	{attribute 'TcIecLibraryType'}
	{attribute 'external_name' := 'F_VN_ImageAverageStdDevExp_GUID_F60066E2_6F02_44CC_C0FB_3753E15EF1D8'}
	(* Computes the (channel-wise) average pixel value and the corresponding standard deviation of an image. (expert function) *)
	FUNCTION F_VN_ImageAverageStdDevExp : HRESULT
	VAR_INPUT
		ipSrcImage	:	ITcVnImage;	(* Source image (1 - 4 channels) *)
	END_VAR
	VAR_IN_OUT
		aAverage	:	TcVnVector4_LREAL;	(* Returns the (channel-wise) average pixel value of ipSrcImage *)
		aStdDev	:	TcVnVector4_LREAL;	(* Returns the (channel-wise) pixel value standard deviation of ipSrcImage *)
	END_VAR
	VAR_INPUT
		ipMask	:	ITcVnImage;	(* Mask of type USINT (1 channel) *)
		hrPrev	:	HRESULT;	(* HRESULT indicating the result of previous operations (If SUCCEEDED(hrPrev) equals false, no operation is executed.) *)
	END_VAR

END_FUNCTION

// Functions/Image Analysis/F_VN_ImageCenterOfMass

	{attribute 'TcIecLibraryType'}
	{attribute 'external_name' := 'F_VN_ImageCenterOfMass_GUID_92F451E2_12EA_4476_D35C_66DCB9E907BA'}
	(* Computes the center of mass of an image. *)
	FUNCTION F_VN_ImageCenterOfMass : HRESULT
	VAR_INPUT
		ipSrcImage	:	ITcVnImage;	(* Source image (1 channel) *)
	END_VAR
	VAR_IN_OUT
		aCenterOfMass	:	TcVnPoint2_LREAL;	(* Returns the center of mass of the image *)
	END_VAR
	VAR_INPUT
		hrPrev	:	HRESULT;	(* HRESULT indicating the result of previous operations (If SUCCEEDED(hrPrev) equals false, no operation is executed.) *)
	END_VAR

END_FUNCTION

// Functions/Image Analysis/F_VN_ImageCenterOfMassExp

	{attribute 'TcIecLibraryType'}
	{attribute 'external_name' := 'F_VN_ImageCenterOfMassExp_GUID_2975F517_49B1_4459_C14B_04840D9F0255'}
	(* Computes the center of mass of an image. *)
	FUNCTION F_VN_ImageCenterOfMassExp : HRESULT
	VAR_INPUT
		ipSrcImage	:	ITcVnImage;	(* Source image (1 channel) *)
	END_VAR
	VAR_IN_OUT
		aCenterOfMass	:	TcVnPoint2_LREAL;	(* Returns the center of mass of the image *)
	END_VAR
	VAR_INPUT
		ipMask	:	ITcVnImage;	(* Optional mask (1 channel of type USINT, same width and height as ipSrcImage) *)
		hrPrev	:	HRESULT;	(* HRESULT indicating the result of previous operations (If SUCCEEDED(hrPrev) equals false, no operation is executed.) *)
	END_VAR

END_FUNCTION

// Functions/Image Analysis/F_VN_ImageMedian

	{attribute 'TcIecLibraryType'}
	{attribute 'external_name' := 'F_VN_ImageMedian_GUID_8462A627_DBC4_4874_EF70_B1418DB7E2BB'}
	(* Computes the (approximated, channel-wise) median pixel value of an image. *)
	FUNCTION F_VN_ImageMedian : HRESULT
	VAR_INPUT
		ipSrcImage	:	ITcVnImage;	(* Source image (1 - 4 channels) *)
	END_VAR
	VAR_IN_OUT
		aMedian	:	TcVnVector4_LREAL;	(* Returns the (approximated, channel-wise) median pixel value of ipSrcImage *)
	END_VAR
	VAR_INPUT
		hrPrev	:	HRESULT;	(* HRESULT indicating the result of previous operations (If SUCCEEDED(hrPrev) equals false, no operation is executed.) *)
	END_VAR

END_FUNCTION

// Functions/Image Analysis/F_VN_ImageMedianExp

	{attribute 'TcIecLibraryType'}
	{attribute 'external_name' := 'F_VN_ImageMedianExp_GUID_04A4F1B3_1CC2_4D44_C68C_989FB7E7D270'}
	(* Computes the (approximated, channel-wise) median pixel value of an image. (expert function) *)
	FUNCTION F_VN_ImageMedianExp : HRESULT
	VAR_INPUT
		ipSrcImage	:	ITcVnImage;	(* Source image (1 - 4 channels) *)
	END_VAR
	VAR_IN_OUT
		aMedian	:	TcVnVector4_LREAL;	(* Returns the (approximated, channel-wise) median pixel value of ipSrcImage *)
	END_VAR
	VAR_INPUT
		ipMask	:	ITcVnImage;	(* Mask of type USINT (1 channel) *)
		hrPrev	:	HRESULT;	(* HRESULT indicating the result of previous operations (If SUCCEEDED(hrPrev) equals false, no operation is executed.) *)
	END_VAR

END_FUNCTION

// Functions/Image Analysis/F_VN_ImageMoments

	{attribute 'TcIecLibraryType'}
	{attribute 'external_name' := 'F_VN_ImageMoments_GUID_967E76E1_3BDD_4152_E4CB_6D63F11261EF'}
	(* Computes the spatial moments, the central moments, and the central normalized moments of an image up to the third order. *)
	FUNCTION F_VN_ImageMoments : HRESULT
	VAR_INPUT
		ipImage	:	ITcVnImage;	(* Source image (1 channel, elements of type USINT or REAL) *)
	END_VAR
	VAR_IN_OUT
		stMoments	:	TcVnMoments;	(* Returns a struct containing the moments *)
	END_VAR
	VAR_INPUT
		bBinaryImage	:	BOOL;	(* If true, all non-zero pixels are treated as ones *)
		hrPrev	:	HRESULT;	(* HRESULT indicating the result of previous operations (If SUCCEEDED(hrPrev) equals false, no operation is executed.) *)
	END_VAR

END_FUNCTION

// Functions/Image Analysis/F_VN_MaxPixelValue

	{attribute 'TcIecLibraryType'}
	{attribute 'external_name' := 'F_VN_MaxPixelValue_GUID_413B82D5_F755_40D2_D677_A4C5ED7EF55F'}
	(* Finds the maximum pixel value in an image (1 - 4 channels supported). *)
	FUNCTION F_VN_MaxPixelValue : HRESULT
	VAR_INPUT
		ipImage	:	ITcVnImage;	(* Source image *)
	END_VAR
	VAR_IN_OUT
		aMaxValue	:	TcVnVector4_LREAL;	(* Returns the maximum pixel value *)
		aPosition	:	TcVnPoint2_DINT;	(* Returns the first found position of aMaxValue *)
	END_VAR
	VAR_INPUT
		hrPrev	:	HRESULT;	(* HRESULT indicating the result of previous operations (If SUCCEEDED(hrPrev) equals false, no operation is executed.) *)
	END_VAR

END_FUNCTION

// Functions/Image Analysis/F_VN_MaxPixelValueExp

	{attribute 'TcIecLibraryType'}
	{attribute 'external_name' := 'F_VN_MaxPixelValueExp_GUID_6DE06A3E_73A8_4932_DDB7_AC3625332A92'}
	(* Finds the maximum pixel value in an image (1 - 4 channels supported). (expert function) *)
	FUNCTION F_VN_MaxPixelValueExp : HRESULT
	VAR_INPUT
		ipImage	:	ITcVnImage;	(* Source image *)
	END_VAR
	VAR_IN_OUT
		aMaxValue	:	TcVnVector4_LREAL;	(* Returns the maximum pixel value *)
		aPosition	:	TcVnPoint2_DINT;	(* Returns the first found position of aMaxValue (not supported for multi-channel images with ELEMENTWISE) *)
	END_VAR
	VAR_INPUT
		ipMask	:	ITcVnImage;	(* Optional mask to specify which pixel positions are considered (USINT, set parameter to 0 if not required) *)
		eVectorCompareMethod	:	ETcVnVectorCompareMethod;	(* Select a vector compare method for multi-channel images *)
		hrPrev	:	HRESULT;	(* HRESULT indicating the result of previous operations (If SUCCEEDED(hrPrev) equals false, no operation is executed.) *)
	END_VAR

END_FUNCTION

// Functions/Image Analysis/F_VN_MinPixelValue

	{attribute 'TcIecLibraryType'}
	{attribute 'external_name' := 'F_VN_MinPixelValue_GUID_2CD718DC_24E2_49FF_F186_BB52705C26CA'}
	(* Finds the minimum pixel value in an image (1 - 4 channels supported). *)
	FUNCTION F_VN_MinPixelValue : HRESULT
	VAR_INPUT
		ipImage	:	ITcVnImage;	(* Source image *)
	END_VAR
	VAR_IN_OUT
		aMinValue	:	TcVnVector4_LREAL;	(* Returns the minimum pixel value *)
		aPosition	:	TcVnPoint2_DINT;	(* Returns the first found position of aMinValue *)
	END_VAR
	VAR_INPUT
		hrPrev	:	HRESULT;	(* HRESULT indicating the result of previous operations (If SUCCEEDED(hrPrev) equals false, no operation is executed.) *)
	END_VAR

END_FUNCTION

// Functions/Image Analysis/F_VN_MinPixelValueExp

	{attribute 'TcIecLibraryType'}
	{attribute 'external_name' := 'F_VN_MinPixelValueExp_GUID_F4A5D3CA_6503_48EC_C514_4486EF0B3DEE'}
	(* Finds the minimum pixel value in an image (1 - 4 channels supported). (expert function) *)
	FUNCTION F_VN_MinPixelValueExp : HRESULT
	VAR_INPUT
		ipImage	:	ITcVnImage;	(* Source image *)
	END_VAR
	VAR_IN_OUT
		aMinValue	:	TcVnVector4_LREAL;	(* Returns the minimum pixel value *)
		aPosition	:	TcVnPoint2_DINT;	(* Returns the first found position of aMinValue (not supported for multi-channel images with ELEMENTWISE) *)
	END_VAR
	VAR_INPUT
		ipMask	:	ITcVnImage;	(* Optional mask to specify which pixel positions are considered (USINT, set parameter to 0 if not required) *)
		eVectorCompareMethod	:	ETcVnVectorCompareMethod;	(* Select a vector compare method for multi-channel images *)
		hrPrev	:	HRESULT;	(* HRESULT indicating the result of previous operations (If SUCCEEDED(hrPrev) equals false, no operation is executed.) *)
	END_VAR

END_FUNCTION

// Functions/Image Analysis/F_VN_RegionOrientation

	{attribute 'TcIecLibraryType'}
	{attribute 'external_name' := 'F_VN_RegionOrientation_GUID_40AE352D_EC33_486F_FD9D_BE6F8D8BC7EF'}
	(* Calculate the orientation of a region based on a binary image that contains a non zero value for every pixel in that region. *)
	FUNCTION F_VN_RegionOrientation : HRESULT
	VAR_INPUT
		ipSrcImage	:	ITcVnImage;	(* Source image (1 channel, binary). *)
	END_VAR
	VAR_IN_OUT
		stOrientation	:	TcVnRotatedRectangle;	(* Resulting rotated rectangle, containig center of mass, lenghts of axes, and rotation angle of the region in clockwise direction. *)
	END_VAR
	VAR_INPUT
		hrPrev	:	HRESULT;	(* HRESULT indicating the result of previous operations (If SUCCEEDED(hrPrev) equals false, no operation is executed.) *)
	END_VAR

END_FUNCTION

// Functions/Image Analysis/F_VN_RegionOrientationExp

	{attribute 'TcIecLibraryType'}
	{attribute 'external_name' := 'F_VN_RegionOrientationExp_GUID_5D1BC303_88B3_462A_E97C_3FA0A9CBE9C1'}
	(* Calculate the orientation of a region based on a binary image that contains a non zero value for every pixel in that region. (expert function) *)
	FUNCTION F_VN_RegionOrientationExp : HRESULT
	VAR_INPUT
		ipSrcImage	:	ITcVnImage;	(* Source image (1 channel, binary) *)
	END_VAR
	VAR_IN_OUT
		stOrientation	:	TcVnRotatedRectangle;	(* Resulting rotated rectangle, containig center of mass, lenghts of axes, and rotation angle of the region in clockwise direction. *)
	END_VAR
	VAR_INPUT
		eMethod	:	ETcVnOrientationMethod;	(* Method for calculating the orientation. *)
		hrPrev	:	HRESULT;	(* HRESULT indicating the result of previous operations (If SUCCEEDED(hrPrev) equals false, no operation is executed.) *)
	END_VAR

END_FUNCTION

// Functions/Image Analysis/F_VN_UprightInnerRectangle

	{attribute 'TcIecLibraryType'}
	{attribute 'external_name' := 'F_VN_UprightInnerRectangle_GUID_EAF07AE8_844F_488F_C920_29FB31213543'}
	(* Computes the maximum area upright inner rectangle inside an area. If the valid area contains very small invalid areas or the performance is too slow, use the expert variant of this function and manually choose a suitable nDownScaleFactor. *)
	FUNCTION F_VN_UprightInnerRectangle : HRESULT
	VAR_INPUT
		ipSrcImage	:	ITcVnImage;	(* Source image (USINT, 1 channel, binary, values > 0 mark valid area) *)
	END_VAR
	VAR_IN_OUT
		stRectangle	:	TcVnRectangle_DINT;	(* Returns the maximum area upright inner rectangle *)
	END_VAR
	VAR_INPUT
		hrPrev	:	HRESULT;	(* HRESULT indicating the result of previous operations (If SUCCEEDED(hrPrev) equals false, no operation is executed.) *)
	END_VAR

END_FUNCTION

// Functions/Image Analysis/F_VN_UprightInnerRectangleExp

	{attribute 'TcIecLibraryType'}
	{attribute 'external_name' := 'F_VN_UprightInnerRectangleExp_GUID_F66C1F20_B07B_43D3_EFEB_2BB901924B64'}
	(* Computes the maximum area upright inner rectangle inside an area. (expert function) *)
	FUNCTION F_VN_UprightInnerRectangleExp : HRESULT
	VAR_INPUT
		ipSrcImage	:	ITcVnImage;	(* Source image (USINT, 1 channel, binary, values > 0 mark valid area) *)
	END_VAR
	VAR_IN_OUT
		stRectangle	:	TcVnRectangle_DINT;	(* Returns the maximum area upright inner rectangle *)
	END_VAR
	VAR_INPUT
		nDownScaleFactor	:	DINT;	(* To tradeoff performance vs. accuracy, a factor can be provided, to reduce the internally used image resolution. As long as invalid areas enclosed in the valid area are larger than nDownScaleFactor, the result usually still is the optimal one. Use -1 to auto select depending on ipSrcImage resolution, 0 to always use full resolution (slower but always optimal result). *)
		hrPrev	:	HRESULT;	(* HRESULT indicating the result of previous operations (If SUCCEEDED(hrPrev) equals false, no operation is executed.) *)
	END_VAR

END_FUNCTION

// Functions/Measurement/F_VN_AdjustSearchWindowOrientationToLinearEdge

	{attribute 'TcIecLibraryType'}
	{attribute 'external_name' := 'F_VN_AdjustSearchWindowOrientationToLinearEdge_GUID_A48BF075_5CF2_441E_E9FD_FC6EEED751A9'}
	(* Adjust the search window to be orthogonal to a linear edge. Might be helpful before calling edge localization and distance measurement functions that rely on the search window. *)
	FUNCTION F_VN_AdjustSearchWindowOrientationToLinearEdge : HRESULT
	VAR_INPUT
		ipSrcImage	:	ITcVnImage;	(* Source image *)
	END_VAR
	VAR_IN_OUT
		aStartPoint	:	TcVnPoint2_REAL;	(* Position from which to start the search process (in the direction of aEndPoint), which is not changed *)
		aEndPoint	:	TcVnPoint2_REAL;	(* Position where the search process ends, which is adjusted by this function *)
	END_VAR
	VAR_INPUT
		eEdgeDirection	:	ETcVnEdgeDirection;	(* Specification of the edge direction to search for *)
		fMinStrength	:	REAL;	(* Specification of the minimum strength (intensity difference) of the edge to search for *)
		nMaxThickness	:	UDINT;	(* Specification of the maximum thickness of the edge to search for, which means fMinStrength must be reached within nMaxThickness pixels *)
		nSearchLines	:	UDINT;	(* Width of the search window, i.e. the number of search lines (3, 5, 7, ...), centered around the line specified by aStartPoint and aEndPoint *)
		hrPrev	:	HRESULT;	(* HRESULT indicating the result of previous operations (If SUCCEEDED(hrPrev) equals false, no operation is executed.) *)
	END_VAR

END_FUNCTION

// Functions/Measurement/F_VN_ClosestPointsBF

	{attribute 'TcIecLibraryType'}
	{attribute 'external_name' := 'F_VN_ClosestPointsBF_GUID_1707A941_3B60_480D_D558_A72227DF9CAA'}
	(* Find the closest distance between two 2d point sets of the same type, using a brute force approach. *)
	FUNCTION F_VN_ClosestPointsBF : HRESULT
	VAR_INPUT
		ipPointSet1	:	ITcVnContainer;	(* Container with 1st set of 2d points *)
		ipPointSet2	:	ITcVnContainer;	(* Container with 2nd set of 2d points *)
	END_VAR
	VAR_IN_OUT
		fMinDist	:	LREAL;	(* Returns the minimum distance between 2 points of the different point sets *)
		aPoint1	:	TcVnPoint2_LREAL;	(* Returns the point out of ipPointSet1, for which fMinDist is achieved *)
		aPoint2	:	TcVnPoint2_LREAL;	(* Returns the point out of ipPointSet2, for which fMinDist is achieved *)
	END_VAR
	VAR_INPUT
		hrPrev	:	HRESULT;	(* HRESULT indicating the result of previous operations (If SUCCEEDED(hrPrev) equals false, no operation is executed.) *)
	END_VAR

END_FUNCTION

// Functions/Measurement/F_VN_LocateCircularArc

	{attribute 'TcIecLibraryType'}
	{attribute 'external_name' := 'F_VN_LocateCircularArc_GUID_B3EA520B_4A30_4994_E483_8C5CDCF1D071'}
	(* Locate a circular arc, using an interpolation method. *)
	FUNCTION F_VN_LocateCircularArc : HRESULT
	VAR_INPUT
		ipSrcImage	:	ITcVnImage;	(* Source image (1 channel) *)
	END_VAR
	VAR_IN_OUT
		stCircularArc	:	TcVnCircularArc;	(* Returns the circular arc parameters *)
		aCenter	:	TcVnPoint2_REAL;	(* Input estimated circle center (only used as a starting point to search for the circle contour, not used for the circle center estimation) *)
	END_VAR
	VAR_INPUT
		fSearchRadius	:	REAL;	(* Input search radius (starting from aCenter, should be greater than the actual circle radius but aCenter + fSearchRadius should be within the image borders) *)
		fArcDirectionRad	:	LREAL;	(* Input search starting direction in radian. Valid range is [-pi, +pi], where right is 0 rad, top is -pi/2 rad and bottom +pi/2 rad. The circular arc should at least be valid in range fArcDirectionRad +- 0.4 rad. *)
		eEdgeDirection	:	ETcVnEdgeDirection;	(* Specification of the edge direction to search for *)
		fMinStrength	:	REAL;	(* Specification of the minimum strength (intensity difference) of the edge to search for *)
		hrPrev	:	HRESULT;	(* HRESULT indicating the result of previous operations (If SUCCEEDED(hrPrev) equals false, no operation is executed.) *)
	END_VAR

END_FUNCTION

// Functions/Measurement/F_VN_LocateCircularArcExp

	{attribute 'TcIecLibraryType'}
	{attribute 'external_name' := 'F_VN_LocateCircularArcExp_GUID_3DE4C842_0688_45E4_D1B3_D06158B1C008'}
	(* Locate a circular arc. (expert function) *)
	FUNCTION F_VN_LocateCircularArcExp : HRESULT
	VAR_INPUT
		ipSrcImage	:	ITcVnImage;	(* Source image (1 channel) *)
	END_VAR
	VAR_IN_OUT
		stCircularArc	:	TcVnCircularArc;	(* Returns the circular arc parameters *)
		aCenter	:	TcVnPoint2_REAL;	(* Input estimated circle center (only used as a starting point to search for the circle contour, not used for the circle center estimation) *)
	END_VAR
	VAR_INPUT
		fSearchRadius	:	REAL;	(* Input search radius (starting from aCenter, should be greater than the actual circle radius but aCenter + fSearchRadius should be within the image borders) *)
		fArcDirectionRad	:	LREAL;	(* Input search starting direction in radian. Valid range is [-pi, +pi], where right is 0 rad, top is -pi/2 rad and bottom +pi/2 rad. The circular arc should at least be valid in range fArcDirectionRad +- 4 * fAngleStepRad) *)
		eEdgeDirection	:	ETcVnEdgeDirection;	(* Specification of the edge direction to search for *)
		fMinStrength	:	REAL;	(* Specification of the minimum strength (intensity difference) of the edge to search for *)
		fAngleStepRad	:	LREAL;	(* Search step in rad (should be chosen so that about 20 - 60 steps are available for the whole arc. In most cases 0.1 rad (5.7 deg) is a good value) *)
		nMaxThickness	:	UDINT;	(* Specification of the maximum thickness of the edge to search for, which means fMinStrength must be reached within nMaxThickness pixels *)
		bInvertSearchDirection	:	BOOL;	(* If true, the search starts from outside the circular arc in direction of the center *)
		nSubpixelsIterations	:	UDINT;	(* Specifies the number of subpixels (for INTERPOLATION, 10 - 20 usually is sufficient) or maximum number of iterations for optimizing the parameters (for APPROX_ERF and APPROX_GAUSSIAN, 50 - 100 usually is sufficient) *)
		fApproxPrecision	:	REAL;	(* Specifies the approximation precision for APPROX_ERF and APPROX_GAUSSIAN (0.001 usually is sufficient, unused for INTERPOLATION) *)
		eAlgorithm	:	ETcVnEdgeDetectionAlgorithm;	(* Selection of the edge detection algorithm *)
		ipContourPoints	:	REFERENCE TO ITcVnContainer;	(* Returns the subpixel accurate contour (optional, set to 0 if not required; ContainerType_Vector_TcVnPoint2_REAL; Non-zero interface pointers are reused.) *)
		hrPrev	:	HRESULT;	(* HRESULT indicating the result of previous operations (If SUCCEEDED(hrPrev) equals false, no operation is executed.) *)
	END_VAR

END_FUNCTION

// Functions/Measurement/F_VN_LocateEdge

	{attribute 'TcIecLibraryType'}
	{attribute 'external_name' := 'F_VN_LocateEdge_GUID_821673DE_5105_465A_CB38_62BD7B02ED8D'}
	(* Locate the points of the first occuring edge inside a specified search window, using an interpolation method. *)
	FUNCTION F_VN_LocateEdge : HRESULT
	VAR_INPUT
		ipSrcImage	:	ITcVnImage;	(* Source image (1 channel) *)
		ipEdgePoints	:	REFERENCE TO ITcVnContainer;	(* Returns the detected edge points (ContainerType_Vector_TcVnPoint2_REAL) *)
	END_VAR
	VAR_IN_OUT
		aStartPoint	:	TcVnPoint2_REAL;	(* Position from which to start the search process (in the direction of aEndPoint) *)
		aEndPoint	:	TcVnPoint2_REAL;	(* Position where the search process ends *)
	END_VAR
	VAR_INPUT
		eEdgeDirection	:	ETcVnEdgeDirection;	(* Specification of the edge direction to search for *)
		fMinStrength	:	REAL;	(* Specification of the minimum strength (intensity difference) of the edge to search for *)
		nSearchLines	:	UDINT;	(* Width of the search window, i.e. the number of search lines (1, 3, 5, 7, ...), centered around the line specified by aStartPoint and aEndPoint *)
		hrPrev	:	HRESULT;	(* HRESULT indicating the result of previous operations (If SUCCEEDED(hrPrev) equals false, no operation is executed.) *)
	END_VAR
	VAR_OUTPUT
		fAvgStrength	:	REAL;	(* Returns the average strength of the detected edge *)
	END_VAR

END_FUNCTION

// Functions/Measurement/F_VN_LocateEdgeExp

	{attribute 'TcIecLibraryType'}
	{attribute 'external_name' := 'F_VN_LocateEdgeExp_GUID_9EF58615_240A_46AE_FF21_3A1E56AF0C88'}
	(* Locate the points of the first occuring edge inside a specified search window with subpixel accuracy. (expert function) *)
	FUNCTION F_VN_LocateEdgeExp : HRESULT
	VAR_INPUT
		ipSrcImage	:	ITcVnImage;	(* Source image (1 channel) *)
		ipEdgePoints	:	REFERENCE TO ITcVnContainer;	(* Returns the detected edge points (ContainerType_Vector_TcVnPoint2_REAL) *)
	END_VAR
	VAR_IN_OUT
		aStartPoint	:	TcVnPoint2_REAL;	(* Position from which to start the search process (in the direction of aEndPoint) *)
		aEndPoint	:	TcVnPoint2_REAL;	(* Position where the search process ends *)
	END_VAR
	VAR_INPUT
		eEdgeDirection	:	ETcVnEdgeDirection;	(* Specification of the edge direction to search for *)
		fMinStrength	:	REAL;	(* Specification of the minimum strength (intensity difference) of the edge to search for *)
		nSearchLines	:	UDINT;	(* Width of the search window, i.e. the number of search lines (1, 3, 5, 7, ...), centered around the line specified by aStartPoint and aEndPoint *)
		fSearchLineDist	:	REAL;	(* Distance between the search lines in pixels (> 0) *)
		nMaxThickness	:	UDINT;	(* Specification of the maximum thickness of the edge to search for, which means fMinStrength must be reached within nMaxThickness pixels *)
		nSubpixelsIterations	:	UDINT;	(* Specifies the number of subpixels (for INTERPOLATION, 10 - 20 usually is sufficient) or maximum number of iterations for optimizing the parameters (for APPROX_ERF and APPROX_GAUSSIAN, 50 - 100 usually is sufficient) *)
		fApproxPrecision	:	REAL;	(* Specifies the approximation precision for APPROX_ERF and APPROX_GAUSSIAN (0.001 usually is sufficient, unused for INTERPOLATION) *)
		eAlgorithm	:	ETcVnEdgeDetectionAlgorithm;	(* Selection of the edge detection algorithm *)
		hrPrev	:	HRESULT;	(* HRESULT indicating the result of previous operations (If SUCCEEDED(hrPrev) equals false, no operation is executed.) *)
	END_VAR
	VAR_OUTPUT
		fAvgStrength	:	REAL;	(* Returns the average strength of the detected edge *)
	END_VAR

END_FUNCTION

// Functions/Measurement/F_VN_LocateEdges

	{attribute 'TcIecLibraryType'}
	{attribute 'external_name' := 'F_VN_LocateEdges_GUID_F9BEA670_3E7B_41AF_C134_87CCD25817E5'}
	(* Locate the points of multiple occuring edges inside a specified search window, using an interpolation method. *)
	FUNCTION F_VN_LocateEdges : HRESULT
	VAR_INPUT
		ipSrcImage	:	ITcVnImage;	(* Source image (1 channel) *)
		ipEdgePoints	:	REFERENCE TO ITcVnContainer;	(* Returns the detected edge points (ContainerType_Vector_Vector_TcVnPoint2_REAL) *)
	END_VAR
	VAR_IN_OUT
		aStartPoint	:	TcVnPoint2_REAL;	(* Position from which to start the search process (in the direction of aEndPoint) *)
		aEndPoint	:	TcVnPoint2_REAL;	(* Position where the search process ends *)
	END_VAR
	VAR_INPUT
		nNumEdges	:	UDINT;	(* The (maximum) number of edges to search for *)
		eEdgeDirection	:	ETcVnEdgeDirection;	(* Specification of the edge direction to search for *)
		bAlternateDirection	:	BOOL;	(* If true, eEdgeDirection is alternated after each detected edge. Else, only edges with eEdgeDirection are searched for. *)
		fMinStrength	:	REAL;	(* Specification of the minimum strength (intensity difference) of the edge to search for *)
		nSearchLines	:	UDINT;	(* Width of the search window, i.e. the number of search lines (1, 3, 5, 7, ...), centered around the line specified by aStartPoint and aEndPoint *)
		hrPrev	:	HRESULT;	(* HRESULT indicating the result of previous operations (If SUCCEEDED(hrPrev) equals false, no operation is executed.) *)
	END_VAR
	VAR_OUTPUT
		fAvgStrength	:	REAL;	(* Returns the average strength of the detected edges *)
	END_VAR

END_FUNCTION

// Functions/Measurement/F_VN_LocateEdgesExp

	{attribute 'TcIecLibraryType'}
	{attribute 'external_name' := 'F_VN_LocateEdgesExp_GUID_CBD8E9BC_8404_4662_FBC2_518D80CA7608'}
	(* Locate the points of multiple occuring edges inside a specified search window with subpixel accuracy. (expert function) *)
	FUNCTION F_VN_LocateEdgesExp : HRESULT
	VAR_INPUT
		ipSrcImage	:	ITcVnImage;	(* Source image (1 channel) *)
		ipEdgePoints	:	REFERENCE TO ITcVnContainer;	(* Returns the detected edge points (ContainerType_Vector_Vector_TcVnPoint2_REAL) *)
	END_VAR
	VAR_IN_OUT
		aStartPoint	:	TcVnPoint2_REAL;	(* Position from which to start the search process (in the direction of aEndPoint) *)
		aEndPoint	:	TcVnPoint2_REAL;	(* Position where the search process ends *)
	END_VAR
	VAR_INPUT
		nNumEdges	:	UDINT;	(* The (maximum) number of edges to search for *)
		eEdgeDirection	:	ETcVnEdgeDirection;	(* Specification of the edge direction to search for *)
		bAlternateDirection	:	BOOL;	(* If true, eEdgeDirection is alternated after each detected edge. Else, only edges with eEdgeDirection are searched for. *)
		fMinStrength	:	REAL;	(* Specification of the minimum strength (intensity difference) of the edge to search for *)
		nSearchLines	:	UDINT;	(* Width of the search window, i.e. the number of search lines (1, 3, 5, 7, ...), centered around the line specified by aStartPoint and aEndPoint *)
		fSearchLineDist	:	REAL;	(* Distance between the search lines in pixels (> 0) *)
		nMaxThickness	:	UDINT;	(* Specification of the maximum thickness of the edge to search for, which means fMinStrength must be reached within nMaxThickness pixels *)
		nSubpixelsIterations	:	UDINT;	(* Specifies the number of subpixels (for INTERPOLATION, 10 - 20 usually is sufficient) or maximum number of iterations for optimizing the parameters (for APPROX_ERF and APPROX_GAUSSIAN, 50 - 100 usually is sufficient) *)
		fApproxPrecision	:	REAL;	(* Specifies the approximation precision for APPROX_ERF and APPROX_GAUSSIAN (0.001 usually is sufficient, unused for INTERPOLATION) *)
		eAlgorithm	:	ETcVnEdgeDetectionAlgorithm;	(* Selection of the edge detection algorithm *)
		hrPrev	:	HRESULT;	(* HRESULT indicating the result of previous operations (If SUCCEEDED(hrPrev) equals false, no operation is executed.) *)
	END_VAR
	VAR_OUTPUT
		fAvgStrength	:	REAL;	(* Returns the average strength of the detected edges *)
	END_VAR

END_FUNCTION

// Functions/Measurement/F_VN_LocateEllipse

	{attribute 'TcIecLibraryType'}
	{attribute 'external_name' := 'F_VN_LocateEllipse_GUID_9220076D_04F4_4060_F21C_5859876A1EAA'}
	(* Locate an ellipse, using an interpolation method for locating the edges. *)
	FUNCTION F_VN_LocateEllipse : HRESULT
	VAR_INPUT
		ipSrcImage	:	ITcVnImage;	(* Source image (1 channel) *)
	END_VAR
	VAR_IN_OUT
		stEllipse	:	TcVnRotatedRectangle;	(* Returns the detected ellipse *)
		aCenter	:	TcVnPoint2_REAL;	(* The expected ellipse center *)
	END_VAR
	VAR_INPUT
		fSearchRadius	:	REAL;	(* Radius around aCenter to search for edges (aCenter + fSearchRadius in all directions must be inside image borders!) *)
		eEdgeDirection	:	ETcVnEdgeDirection;	(* Specification of the edge direction to search for (from center to outside ellipse) *)
		fMinStrength	:	REAL;	(* Specification of the minimum strength (intensity difference) of the edge to search for *)
		hrPrev	:	HRESULT;	(* HRESULT indicating the result of previous operations (If SUCCEEDED(hrPrev) equals false, no operation is executed.) *)
	END_VAR

END_FUNCTION

// Functions/Measurement/F_VN_LocateEllipseExp

	{attribute 'TcIecLibraryType'}
	{attribute 'external_name' := 'F_VN_LocateEllipseExp_GUID_E51341EF_78F5_4F0B_EFBC_F53D28C9F2F9'}
	(* Locate an ellipse. (expert function) *)
	FUNCTION F_VN_LocateEllipseExp : HRESULT
	VAR_INPUT
		ipSrcImage	:	ITcVnImage;	(* Source image (1 channel) *)
	END_VAR
	VAR_IN_OUT
		stEllipse	:	TcVnRotatedRectangle;	(* Returns the detected ellipse *)
		aCenter	:	TcVnPoint2_REAL;	(* The expected ellipse center *)
	END_VAR
	VAR_INPUT
		fSearchRadius	:	REAL;	(* Radius around aCenter to search for edges *)
		eEdgeDirection	:	ETcVnEdgeDirection;	(* Specification of the edge direction to search for (from center to outside ellipse or other way round, if bInvertSearchDirection is true) *)
		fMinStrength	:	REAL;	(* Specification of the minimum strength (intensity difference) of the edge to search for *)
		nMaxThickness	:	UDINT;	(* Specification of the maximum thickness of the edge to search for, which means fMinStrength must be reached within nMaxThickness pixels *)
		bInvertSearchDirection	:	BOOL;	(* If true, the search starts from outside the ellipse in direction of the center *)
		fMinSearchRadius	:	REAL;	(* Radius around aCenter to skip before starting to search for edges (e.g. to save time or if the center contains edges that should be ignored) *)
		nSubpixelsIterations	:	UDINT;	(* Specifies the number of subpixels (for INTERPOLATION, 10 - 20 usually is sufficient) or maximum number of iterations for optimizing the parameters (for APPROX_ERF and APPROX_GAUSSIAN, 50 - 100 usually is sufficient) *)
		nSearchLines	:	UDINT;	(* Specifies the amount of search lines, which are equally distributed in all directions (must be >= 8 and a multiple of 4) *)
		fApproxPrecision	:	REAL;	(* Specifies the approximation precision for APPROX_ERF and APPROX_GAUSSIAN (0.001 usually is sufficient, unused for INTERPOLATION) *)
		eAlgorithm	:	ETcVnEdgeDetectionAlgorithm;	(* Selection of the edge detection algorithm *)
		ipContourPoints	:	REFERENCE TO ITcVnContainer;	(* Returns the subpixel accurate ellipse contour (optional, set to 0 if not required; ContainerType_Vector_TcVnPoint2_REAL; Non-zero interface pointers are reused.) *)
		hrPrev	:	HRESULT;	(* HRESULT indicating the result of previous operations (If SUCCEEDED(hrPrev) equals false, no operation is executed.) *)
	END_VAR

END_FUNCTION

// Functions/Measurement/F_VN_MeasureAngleBetweenEdges

	{attribute 'TcIecLibraryType'}
	{attribute 'external_name' := 'F_VN_MeasureAngleBetweenEdges_GUID_3F365496_F29D_4CB2_E29C_22AFE1946B81'}
	(* Measure the angle between 2 edges, using an interpolation method. *)
	FUNCTION F_VN_MeasureAngleBetweenEdges : HRESULT
	VAR_INPUT
		ipSrcImage	:	ITcVnImage;	(* Source image (1 channel) *)
	END_VAR
	VAR_IN_OUT
		fAngle	:	REAL;	(* Returns the angle between the detected edges (radians) *)
		aInnerPoint	:	TcVnPoint2_REAL;	(* Position inside the angle to measure, from which to start the edge search process (in the direction of aOuterPoint1 and aOuterPoint2) *)
		aOuterPoint1	:	TcVnPoint2_REAL;	(* Position where the search process for edge 1 ends *)
		aOuterPoint2	:	TcVnPoint2_REAL;	(* Position where the search process for edge 2 ends *)
	END_VAR
	VAR_INPUT
		eEdgeDirection	:	ETcVnEdgeDirection;	(* Specification of the edge direction from aInnerPoint to aOuterPoint1 and aOuterPoint2 to search for *)
		fMinStrength	:	REAL;	(* Specification of the minimum strength (intensity difference) of the edge to search for *)
		nSearchLines	:	UDINT;	(* Width of the search windows, i.e. the number of search lines (3, 5, 7, ...), centered around the lines specified by aInnerPoint and aOuterPoint1, aOuterPoint2 *)
		hrPrev	:	HRESULT;	(* HRESULT indicating the result of previous operations (If SUCCEEDED(hrPrev) equals false, no operation is executed.) *)
	END_VAR

END_FUNCTION

// Functions/Measurement/F_VN_MeasureAngleBetweenEdgesExp

	{attribute 'TcIecLibraryType'}
	{attribute 'external_name' := 'F_VN_MeasureAngleBetweenEdgesExp_GUID_568F7F67_1C70_4FED_D486_E63C419ABA30'}
	(* Measure the angle between 2 edges. *)
	FUNCTION F_VN_MeasureAngleBetweenEdgesExp : HRESULT
	VAR_INPUT
		ipSrcImage	:	ITcVnImage;	(* Source image (1 channel) *)
	END_VAR
	VAR_IN_OUT
		fAngle	:	REAL;	(* Returns the angle between the detected edges (radians or degrees, depending on bAngleInDegrees) *)
		aInnerPoint	:	TcVnPoint2_REAL;	(* Position inside the angle to measure, from which to start the edge search process (in the direction of aOuterPoint1 and aOuterPoint2) *)
		aOuterPoint1	:	TcVnPoint2_REAL;	(* Position where the search process for edge 1 ends *)
		aOuterPoint2	:	TcVnPoint2_REAL;	(* Position where the search process for edge 2 ends *)
	END_VAR
	VAR_INPUT
		eEdgeDirection	:	ETcVnEdgeDirection;	(* Specification of the edge direction from aInnerPoint to aOuterPoint1 and aOuterPoint2 to search for *)
		fMinStrength	:	REAL;	(* Specification of the minimum strength (intensity difference) of the edge to search for *)
		nSearchLines	:	UDINT;	(* Width of the search window, i.e. the number of search lines (3, 5, 7, ...), centered around the line specified by aInnerPoint and aOuterPoint1, aOuterPoint2 *)
		fSearchLineDist	:	REAL;	(* Distance between the search lines in pixels (> 0) *)
		nMaxThickness	:	UDINT;	(* Specification of the maximum thickness of the edge to search for, which means fMinStrength must be reached within nMaxThickness pixels *)
		bInvertSearchDirection	:	BOOL;	(* If true, the search starts from each aOuterPoint in direction of aInnerPoint *)
		nSubpixelsIterations	:	UDINT;	(* Specifies the number of subpixels (for INTERPOLATION, 10 - 20 usually is sufficient) or maximum number of iterations for optimizing the parameters (for APPROX_ERF and APPROX_GAUSSIAN, 50 - 100 usually is sufficient) *)
		bAngleInDegrees	:	BOOL;	(* fAngle is in degrees, if true *)
		fApproxPrecision	:	REAL;	(* Specifies the approximation precision for APPROX_ERF and APPROX_GAUSSIAN (0.001 usually is sufficient, unused for INTERPOLATION) *)
		eAlgorithm	:	ETcVnEdgeDetectionAlgorithm;	(* Selection of the edge detection algorithm *)
		ipEdgePoints1	:	REFERENCE TO ITcVnContainer;	(* Returns the detected edge points between aInnerPoint and aOuterPoint1 (ContainerType_Vector_TcVnPoint2_REAL) *)
		ipEdgePoints2	:	REFERENCE TO ITcVnContainer;	(* Returns the detected edge points between aInnerPoint and aOuterPoint2 (ContainerType_Vector_TcVnPoint2_REAL) *)
		hrPrev	:	HRESULT;	(* HRESULT indicating the result of previous operations (If SUCCEEDED(hrPrev) equals false, no operation is executed.) *)
	END_VAR

END_FUNCTION

// Functions/Measurement/F_VN_MeasureEdgeDistance

	{attribute 'TcIecLibraryType'}
	{attribute 'external_name' := 'F_VN_MeasureEdgeDistance_GUID_8442B5B8_5621_45A5_E95E_AE93563506B4'}
	(* Measure the distance between 2 parallel edges, using an interpolation method. *)
	FUNCTION F_VN_MeasureEdgeDistance : HRESULT
	VAR_INPUT
		ipSrcImage	:	ITcVnImage;	(* Source image (1 channel) *)
	END_VAR
	VAR_IN_OUT
		fAvgDistance	:	REAL;	(* Returns the average distance between the detected edges *)
		aStartPoint	:	TcVnPoint2_REAL;	(* Position from which to start the search process (in the direction of aEndPoint) *)
		aEndPoint	:	TcVnPoint2_REAL;	(* Position where the search process ends *)
	END_VAR
	VAR_INPUT
		eEdgeDirection	:	ETcVnEdgeDirection;	(* Specification of the edge direction from aStartPoint to aEndPoint to search for *)
		fMinStrength	:	REAL;	(* Specification of the minimum strength (intensity difference) of the edge to search for *)
		nSearchLines	:	UDINT;	(* Width of the search window, i.e. the number of search lines (1, 3, 5, 7, ...), centered around the line specified by aStartPoint and aEndPoint *)
		hrPrev	:	HRESULT;	(* HRESULT indicating the result of previous operations (If SUCCEEDED(hrPrev) equals false, no operation is executed.) *)
	END_VAR

END_FUNCTION

// Functions/Measurement/F_VN_MeasureEdgeDistanceExp

	{attribute 'TcIecLibraryType'}
	{attribute 'external_name' := 'F_VN_MeasureEdgeDistanceExp_GUID_5AD56682_D8B6_4B0F_E56F_EECEA1B1D30D'}
	(* Measure the distance between 2 parallel edges. (expert function) *)
	FUNCTION F_VN_MeasureEdgeDistanceExp : HRESULT
	VAR_INPUT
		ipSrcImage	:	ITcVnImage;	(* Source image (1 channel) *)
	END_VAR
	VAR_IN_OUT
		fAvgDistance	:	REAL;	(* Returns the average distance between the detected edges *)
		aStartPoint	:	TcVnPoint2_REAL;	(* Position from which to start the search process (in the direction of aEndPoint) *)
		aEndPoint	:	TcVnPoint2_REAL;	(* Position where the search process ends *)
	END_VAR
	VAR_INPUT
		eEdgeDirection	:	ETcVnEdgeDirection;	(* Specification of the edge direction from aStartPoint to aEndPoint to search for *)
		fMinStrength	:	REAL;	(* Specification of the minimum strength (intensity difference) of the edge to search for *)
		nSearchLines	:	UDINT;	(* Width of the search window, i.e. the number of search lines (1, 3, 5, 7, ...), centered around the line specified by aStartPoint and aEndPoint *)
		fSearchLineDist	:	REAL;	(* Distance between the search lines in pixels (> 0) *)
		nMaxThickness	:	UDINT;	(* Specification of the maximum thickness of the edge to search for, which means fMinStrength must be reached within nMaxThickness pixels *)
		bInvertSearchDirection	:	BOOL;	(* If true, the search starts from the center point between aStartPoint and aEndPoint in both directions *)
		fSearchGap	:	REAL;	(* Optional width of a gap (>= 0, centered between aStartPoint and aEndPoint), that is neglected for searching edges (can reduce execution time). The 2 edges to search for must be on different sides of the gap. *)
		nSubpixelsIterations	:	UDINT;	(* Specifies the number of subpixels (for INTERPOLATION, 10 - 20 usually is sufficient) or maximum number of iterations for optimizing the parameters (for APPROX_ERF and APPROX_GAUSSIAN, 50 - 100 usually is sufficient) *)
		fApproxPrecision	:	REAL;	(* Specifies the approximation precision for APPROX_ERF and APPROX_GAUSSIAN (0.001 usually is sufficient, unused for INTERPOLATION) *)
		eAlgorithm	:	ETcVnEdgeDetectionAlgorithm;	(* Selection of the edge detection algorithm *)
		ipEdgePoints1	:	REFERENCE TO ITcVnContainer;	(* Returns the detected edge points of the edge near aStartPoint (optional, set to 0 if not required; ContainerType_Vector_TcVnPoint2_REAL) *)
		ipEdgePoints2	:	REFERENCE TO ITcVnContainer;	(* Returns the detected edge points of the edge near aEndPoint (optional, set to 0 if not required; ContainerType_Vector_TcVnPoint2_REAL) *)
		ipDistances	:	REFERENCE TO ITcVnContainer;	(* Returns the distances between the detected edge points (optional, set to 0 if not required; ContainerType_Vector_REAL) *)
		hrPrev	:	HRESULT;	(* HRESULT indicating the result of previous operations (If SUCCEEDED(hrPrev) equals false, no operation is executed.) *)
	END_VAR

END_FUNCTION

// Functions/Measurement/F_VN_MeasureMinEdgeDistance

	{attribute 'TcIecLibraryType'}
	{attribute 'external_name' := 'F_VN_MeasureMinEdgeDistance_GUID_4216EB9D_8591_4FD7_E108_339D9A9B2435'}
	(* Measure the minimum distance within the specified search window between 2 edges, using an interpolation method. *)
	FUNCTION F_VN_MeasureMinEdgeDistance : HRESULT
	VAR_INPUT
		ipSrcImage	:	ITcVnImage;	(* Source image (1 channel) *)
	END_VAR
	VAR_IN_OUT
		fMinDistance	:	REAL;	(* Returns the minimum distance between the detected edges *)
		aStartPoint	:	TcVnPoint2_REAL;	(* Position from which to start the search process (in the direction of aEndPoint) *)
		aEndPoint	:	TcVnPoint2_REAL;	(* Position where the search process ends *)
	END_VAR
	VAR_INPUT
		eEdgeDirection	:	ETcVnEdgeDirection;	(* Specification of the edge direction from aStartPoint to aEndPoint to search for *)
		fMinStrength	:	REAL;	(* Specification of the minimum strength (intensity difference) of the edge to search for *)
		nSearchLines	:	UDINT;	(* Width of the search window, i.e. the number of search lines (1, 3, 5, 7, ...), centered around the line specified by aStartPoint and aEndPoint *)
		hrPrev	:	HRESULT;	(* HRESULT indicating the result of previous operations (If SUCCEEDED(hrPrev) equals false, no operation is executed.) *)
	END_VAR

END_FUNCTION

// Functions/Measurement/F_VN_MeasureMinEdgeDistanceExp

	{attribute 'TcIecLibraryType'}
	{attribute 'external_name' := 'F_VN_MeasureMinEdgeDistanceExp_GUID_F4BB7BB4_A75C_4811_EF15_80FEA43A47C2'}
	(* Measure the minimum distance within the specified search window between 2 edges. (expert function) *)
	FUNCTION F_VN_MeasureMinEdgeDistanceExp : HRESULT
	VAR_INPUT
		ipSrcImage	:	ITcVnImage;	(* Source image (1 channel) *)
	END_VAR
	VAR_IN_OUT
		fMinDistance	:	REAL;	(* Returns the minimum distance between the detected edges *)
		aStartPoint	:	TcVnPoint2_REAL;	(* Position from which to start the search process (in the direction of aEndPoint) *)
		aEndPoint	:	TcVnPoint2_REAL;	(* Position where the search process ends *)
	END_VAR
	VAR_INPUT
		eEdgeDirection	:	ETcVnEdgeDirection;	(* Specification of the edge direction from aStartPoint to aEndPoint to search for *)
		fMinStrength	:	REAL;	(* Specification of the minimum strength (intensity difference) of the edge to search for *)
		nSearchLines	:	UDINT;	(* Width of the search window, i.e. the number of search lines (1, 3, 5, 7, ...), centered around the line specified by aStartPoint and aEndPoint *)
		fSearchLineDist	:	REAL;	(* Distance between the search lines in pixels (> 0) *)
		nMaxThickness	:	UDINT;	(* Specification of the maximum thickness of the edge to search for, which means fMinStrength must be reached within nMaxThickness pixels *)
		bInvertSearchDirection	:	BOOL;	(* If true, the search starts from the center point between aStartPoint and aEndPoint in both directions *)
		fSearchGap	:	REAL;	(* Optional width of a gap (>= 0, centered between aStartPoint and aEndPoint), that is neglected for searching edges (can reduce execution time). The 2 edges to search for must be on different sides of the gap. *)
		nSubpixelsIterations	:	UDINT;	(* Specifies the number of subpixels (for INTERPOLATION, 10 - 20 usually is sufficient) or maximum number of iterations for optimizing the parameters (for APPROX_ERF and APPROX_GAUSSIAN, 50 - 100 usually is sufficient) *)
		fApproxPrecision	:	REAL;	(* Specifies the approximation precision for APPROX_ERF and APPROX_GAUSSIAN (0.001 usually is sufficient, unused for INTERPOLATION) *)
		eAlgorithm	:	ETcVnEdgeDetectionAlgorithm;	(* Selection of the edge detection algorithm *)
		ipEdgePoints1	:	REFERENCE TO ITcVnContainer;	(* Returns the detected edge points of the edge near aStartPoint (optional, set to 0 if not required; ContainerType_Vector_TcVnPoint2_REAL) *)
		ipEdgePoints2	:	REFERENCE TO ITcVnContainer;	(* Returns the detected edge points of the edge near aEndPoint (optional, set to 0 if not required; ContainerType_Vector_TcVnPoint2_REAL) *)
	END_VAR
	VAR_IN_OUT
		aPoint1	:	TcVnPoint2_REAL;	(* Returns the point on the edge near aStartPoint, for which the minimum distance is achieved *)
		aPoint2	:	TcVnPoint2_REAL;	(* Returns the point on the edge near aEndPoint, for which the minimum distance is achieved *)
	END_VAR
	VAR_INPUT
		hrPrev	:	HRESULT;	(* HRESULT indicating the result of previous operations (If SUCCEEDED(hrPrev) equals false, no operation is executed.) *)
	END_VAR

END_FUNCTION

// Functions/Basic Container Operations/F_VN_AdvanceIterator

	{attribute 'TcIecLibraryType'}
	{attribute 'external_name' := 'F_VN_AdvanceIterator_GUID_5434BC35_88A7_494D_D67F_166B19F62250'}
	(* Advance an iterator by the specified offset. *)
	FUNCTION F_VN_AdvanceIterator : HRESULT
	VAR_INPUT
		ipIterator	:	ITcVnForwardIterator;	(* Iterator to be advanced *)
		nOffset	:	LINT;	(* Offset, by which ipIterator is advanced *)
		hrPrev	:	HRESULT;	(* HRESULT indicating the result of previous operations (If SUCCEEDED(hrPrev) equals false, no operation is executed.) *)
	END_VAR

END_FUNCTION

// Functions/Basic Container Operations/F_VN_CheckIfEmpty

	{attribute 'TcIecLibraryType'}
	{attribute 'external_name' := 'F_VN_CheckIfEmpty_GUID_0FD6C505_E5F5_42C4_E35B_3D20591B3692'}
	(* Checks if the container is empty. (Alternatively use interface method .CheckIfEmpty.) *)
	FUNCTION F_VN_CheckIfEmpty : HRESULT
	VAR_INPUT
		ipContainer	:	ITcVnContainer;	(* Container *)
		hrPrev	:	HRESULT;	(* HRESULT indicating the result of previous operations (If SUCCEEDED(hrPrev) equals false, no operation is executed.) *)
	END_VAR

END_FUNCTION

// Functions/Basic Container Operations/F_VN_CheckIfIteratorIsAtEnd

	{attribute 'TcIecLibraryType'}
	{attribute 'external_name' := 'F_VN_CheckIfIteratorIsAtEnd_GUID_C83E95B8_608C_4277_F8D3_BC53B4FFAAD1'}
	(* Checks if the iterator points to the past-the-end element. (Alternatively use interface method .CheckIfEnd.) *)
	FUNCTION F_VN_CheckIfIteratorIsAtEnd : HRESULT
	VAR_INPUT
		ipIterator	:	ITcVnForwardIterator;	(* Iterator *)
		hrPrev	:	HRESULT;	(* HRESULT indicating the result of previous operations (If SUCCEEDED(hrPrev) equals false, no operation is executed.) *)
	END_VAR

END_FUNCTION

// Functions/Basic Container Operations/F_VN_ConvertContainerType

	{attribute 'TcIecLibraryType'}
	{attribute 'external_name' := 'F_VN_ConvertContainerType_GUID_F95DA822_884E_459D_D254_815729E9DB4A'}
	(* Converts a container to another type (Struct element types are not supported). *)
	FUNCTION F_VN_ConvertContainerType : HRESULT
	VAR_INPUT
		ipSrcContainer	:	ITcVnContainer;	(* Source container *)
		ipDestContainer	:	REFERENCE TO ITcVnContainer;	(* Returns the converted container *)
		nDestTypeGuid	:	GUID;	(* Specifies the destination container type for the conversion *)
		hrPrev	:	HRESULT;	(* HRESULT indicating the result of previous operations (If SUCCEEDED(hrPrev) equals false, no operation is executed.) *)
	END_VAR

END_FUNCTION

// Functions/Basic Container Operations/F_VN_CopyContainer

	{attribute 'TcIecLibraryType'}
	{attribute 'external_name' := 'F_VN_CopyContainer_GUID_225FF68D_4EE0_465F_CCC0_31CEB055C2A1'}
	(* Copys a container. *)
	FUNCTION F_VN_CopyContainer : HRESULT
	VAR_INPUT
		ipSrcContainer	:	ITcVnContainer;	(* Source container *)
		ipDestContainer	:	REFERENCE TO ITcVnContainer;	(* Destination container (same type ID as ipSrcContainer; Non-zero interface pointers are reused.) *)
		hrPrev	:	HRESULT;	(* HRESULT indicating the result of previous operations (If SUCCEEDED(hrPrev) equals false, no operation is executed.) *)
	END_VAR

END_FUNCTION

// Functions/Basic Container Operations/F_VN_CopyContainerElementsConditional_ITcVnContainer

	{attribute 'TcIecLibraryType'}
	{attribute 'external_name' := 'F_VN_CopyContainerElementsConditional_ITcVnContainer_GUID_D7BA1850_6242_46B8_FD74_B156F6259DDF'}
	(* Copys container elements to a new container, depending on a custom condition. *)
	FUNCTION F_VN_CopyContainerElementsConditional_ITcVnContainer : HRESULT
	VAR_INPUT
		ipSrcContainer	:	ITcVnContainer;	(* Source container *)
		ipDestContainer	:	REFERENCE TO ITcVnContainer;	(* Returns a container with elements, that match the condition *)
		ipConditionFB	:	ITcVnCustomElementCondition_ITcVnContainer;	(* Custom condition *)
		hrPrev	:	HRESULT;	(* HRESULT indicating the result of previous operations (If SUCCEEDED(hrPrev) equals false, no operation is executed.) *)
	END_VAR

END_FUNCTION

// Interfaces/Containers/Function Blocks/ITcVnCustomElementCondition_ITcVnContainer

	(* Offers an interface for a custom condition computed for a container. *)
	{attribute 'c++_compatible'}
	INTERFACE ITcVnCustomElementCondition_ITcVnContainer


(* Evaluates the condition for the container. *)
	{attribute 'c++_compatible'}
	{attribute 'minimal_input_size' := '4'}
	{attribute 'pack_mode' := '4'}
	METHOD Condition : BOOL
	VAR_INPUT
		ipElement : ITcVnContainer;
	END_VAR
END_METHOD

END_INTERFACE

// Functions/Basic Container Operations/F_VN_CopyContainerElementsConditional_ITcVnForwardIterator

	{attribute 'TcIecLibraryType'}
	{attribute 'external_name' := 'F_VN_CopyContainerElementsConditional_ITcVnForwardIterator_GUID_BBA04341_B662_40D5_FA7D_525CFA47EAF7'}
	(* Copys container elements to a new container, depending on a custom condition. *)
	FUNCTION F_VN_CopyContainerElementsConditional_ITcVnForwardIterator : HRESULT
	VAR_INPUT
		ipSrcContainer	:	ITcVnContainer;	(* Source container *)
		ipDestContainer	:	REFERENCE TO ITcVnContainer;	(* Returns a container with elements, that match the condition *)
		ipConditionFB	:	ITcVnCustomElementCondition_ITcVnForwardIterator;	(* Custom condition *)
		hrPrev	:	HRESULT;	(* HRESULT indicating the result of previous operations (If SUCCEEDED(hrPrev) equals false, no operation is executed.) *)
	END_VAR

END_FUNCTION

// Interfaces/Containers/Function Blocks/ITcVnCustomElementCondition_ITcVnForwardIterator

	(* Offers an interface for a custom condition computed for an element represented by an ITcVnForwardIterator. *)
	{attribute 'c++_compatible'}
	INTERFACE ITcVnCustomElementCondition_ITcVnForwardIterator


(* Evaluates the condition for the provided element. *)
	{attribute 'c++_compatible'}
	{attribute 'minimal_input_size' := '4'}
	{attribute 'pack_mode' := '4'}
	METHOD Condition : BOOL
	VAR_INPUT
		ipElement : ITcVnForwardIterator;
	END_VAR
END_METHOD

END_INTERFACE

// Functions/Basic Container Operations/F_VN_CreateContainer

	{attribute 'TcIecLibraryType'}
	{attribute 'external_name' := 'F_VN_CreateContainer_GUID_992F2C5B_DA57_4232_E0CD_3ACBDE7DC582'}
	(* Creates a container with type GUID nTypeGuid and return its container interface. *)
	FUNCTION F_VN_CreateContainer : HRESULT
	VAR_INPUT
		ipContainer	:	REFERENCE TO ITcVnContainer;	(* Returns the created container *)
		nTypeGuid	:	GUID;	(* Type GUID of the container to be created *)
		nElementNum	:	ULINT;	(* Number of elements *)
		hrPrev	:	HRESULT;	(* HRESULT indicating the result of previous operations (If SUCCEEDED(hrPrev) equals false, no operation is executed.) *)
	END_VAR

END_FUNCTION

// Functions/Basic Container Operations/F_VN_CreateContainerFromArray

	{attribute 'TcIecLibraryType'}
	{attribute 'external_name' := 'F_VN_CreateContainerFromArray_GUID_52A76897_10EB_4EC3_C91D_C39F0ACECF43'}
	(* Creates a container with type GUID nTypeGuid, initialize it with provided data and return its container interface. Only supported for basic container types, i.e. not for containers of containers. *)
	FUNCTION F_VN_CreateContainerFromArray : HRESULT
	VAR_INPUT
		pData	:	PVOID;	(* Pointer to the data array. Make sure that the array contains at least nElementNum elements and that the array element type matches the container element type. *)
		ipContainer	:	REFERENCE TO ITcVnContainer;	(* Returns the created container *)
		nTypeGuid	:	GUID;	(* Type GUID of the container to be created *)
		nElementNum	:	ULINT;	(* Number of elements to copy from pData *)
		hrPrev	:	HRESULT;	(* HRESULT indicating the result of previous operations (If SUCCEEDED(hrPrev) equals false, no operation is executed.) *)
	END_VAR

END_FUNCTION

// Functions/Basic Container Operations/F_VN_EraseFromContainer

	{attribute 'TcIecLibraryType'}
	{attribute 'external_name' := 'F_VN_EraseFromContainer_GUID_2E7A1753_1E2D_4D75_EB63_D16A311C9CAB'}
	(* Erase elements from a container. *)
	FUNCTION F_VN_EraseFromContainer : HRESULT
	VAR_INPUT
		ipContainer	:	ITcVnContainer;	(* Container from which to erase elements *)
		nStartIdx	:	ULINT;	(* Index of the first element to erase *)
		nCount	:	ULINT;	(* Number of elements to erase *)
		hrPrev	:	HRESULT;	(* HRESULT indicating the result of previous operations (If SUCCEEDED(hrPrev) equals false, no operation is executed.) *)
	END_VAR

END_FUNCTION

// Functions/Basic Container Operations/F_VN_ExportContainer

	{attribute 'TcIecLibraryType'}
	{attribute 'external_name' := 'F_VN_ExportContainer_GUID_4BEC08A0_88C0_4CBC_DD78_7959C1F8FA73'}
	(* Export the container elements into a buffer (e.g. an array). Only possible for containers with basic elements. *)
	FUNCTION F_VN_ExportContainer : HRESULT
	VAR_INPUT
		ipContainer	:	ITcVnContainer;	(* Container with basic elements *)
		pBuffer	:	PVOID;	(* Buffer to store the container elements (Make sure to allocate enough memory! The required size in bytes can be determined using the function F_VN_ExportContainerSize) *)
		nBufferSize	:	ULINT;	(* Size of the buffer memory in bytes *)
		hrPrev	:	HRESULT;	(* HRESULT indicating the result of previous operations (If SUCCEEDED(hrPrev) equals false, no operation is executed.) *)
	END_VAR

END_FUNCTION

// Functions/Basic Container Operations/F_VN_ExportContainerSize

	{attribute 'TcIecLibraryType'}
	{attribute 'external_name' := 'F_VN_ExportContainerSize_GUID_8E08EEFD_AA9E_43FF_D078_BAF279CFF733'}
	(* Determine the required buffer size in bytes to store all container elements (number_of_Elements * size_per_Element). Only possible for containers with basic elements. *)
	FUNCTION F_VN_ExportContainerSize : HRESULT
	VAR_INPUT
		ipContainer	:	ITcVnContainer;	(* Container with basic elements *)
	END_VAR
	VAR_IN_OUT
		nBufferSize	:	ULINT;	(* Output parameter containing the required buffer size *)
	END_VAR
	VAR_INPUT
		hrPrev	:	HRESULT;	(* HRESULT indicating the result of previous operations (If SUCCEEDED(hrPrev) equals false, no operation is executed.) *)
	END_VAR

END_FUNCTION

// Functions/Basic Container Operations/F_VN_ExportContainer_String

	{attribute 'TcIecLibraryType'}
	{attribute 'external_name' := 'F_VN_ExportContainer_String_GUID_A324FE89_0BFB_42D6_E938_52B6F4BF92D8'}
	(* Export the container elements into a string. Only possible for containers of type ContainerType_String_SINT. *)
	FUNCTION F_VN_ExportContainer_String : HRESULT
	VAR_INPUT
		ipContainer	:	ITcVnContainer;	(* Container of type ContainerType_String_SINT *)
	END_VAR
	VAR_IN_OUT CONSTANT
		sText	:	STRING;	(* Make sure to choose a sufficient STRING size! The required size can be determined using the function VnExportContainerSize. *)
	END_VAR
	VAR_INPUT
		nMaxLength	:	ULINT;	(* Maximum string length to export (including 0 termination). If the container content is longer, the string is cut off at nMaxLength - 1 and 0 termination is appended. In this case, S_FALSE is returned. *)
		hrPrev	:	HRESULT;	(* HRESULT indicating the result of previous operations (If SUCCEEDED(hrPrev) equals false, no operation is executed.) *)
	END_VAR

END_FUNCTION

// Functions/Basic Container Operations/F_VN_ExportSubContainer

	{attribute 'TcIecLibraryType'}
	{attribute 'external_name' := 'F_VN_ExportSubContainer_GUID_D48A84CB_DD40_4E59_FFF5_005B912B1A4A'}
	(* Export the container elements of a sub-container into a buffer (e.g. an array). Only possible for 2-dimensional containers with basic elements. *)
	FUNCTION F_VN_ExportSubContainer : HRESULT
	VAR_INPUT
		ipContainer	:	ITcVnContainer;	(* Container with basic elements *)
		nIndex	:	ULINT;	(* Index of the requested element *)
		pBuffer	:	PVOID;	(* Buffer to store the container elements (Make sure to allocate enough memory! The required size in bytes can be determined using the function F_VN_ExportSubContainerSize) *)
		nBufferSize	:	ULINT;	(* Size of the buffer memory in bytes *)
		hrPrev	:	HRESULT;	(* HRESULT indicating the result of previous operations (If SUCCEEDED(hrPrev) equals false, no operation is executed.) *)
	END_VAR

END_FUNCTION

// Functions/Basic Container Operations/F_VN_ExportSubContainerSize

	{attribute 'TcIecLibraryType'}
	{attribute 'external_name' := 'F_VN_ExportSubContainerSize_GUID_62CBD43B_2ED5_41F9_CEB3_8F27329EC5FA'}
	(* Determine the required buffer size in bytes to store all container elements of a sub-container (number_of_Elements * size_per_Element). Only possible for 2-dimensional containers with basic elements. *)
	FUNCTION F_VN_ExportSubContainerSize : HRESULT
	VAR_INPUT
		ipContainer	:	ITcVnContainer;	(* Container with basic elements *)
		nIndex	:	ULINT;	(* Index of the requested element *)
	END_VAR
	VAR_IN_OUT
		nBufferSize	:	ULINT;	(* Output parameter containing the required buffer size *)
	END_VAR
	VAR_INPUT
		hrPrev	:	HRESULT;	(* HRESULT indicating the result of previous operations (If SUCCEEDED(hrPrev) equals false, no operation is executed.) *)
	END_VAR

END_FUNCTION

// Functions/Basic Container Operations/F_VN_ExportSubContainer_String

	{attribute 'TcIecLibraryType'}
	{attribute 'external_name' := 'F_VN_ExportSubContainer_String_GUID_B7A90F40_E78D_4CCA_CDE5_0E55BDB1D365'}
	(* Export the container elements of a sub-container into a string. Only possible for 2-dimensional containers of type ContainerType_Vector_String_SINT. *)
	FUNCTION F_VN_ExportSubContainer_String : HRESULT
	VAR_INPUT
		ipContainer	:	ITcVnContainer;	(* Container of type ContainerType_Vector_String_SINT *)
		nIndex	:	ULINT;	(* Index of the requested element *)
	END_VAR
	VAR_IN_OUT CONSTANT
		sText	:	STRING;	(* Make sure to choose a sufficient STRING size! The required size can be determined using the function VnExportSubContainerSize. *)
	END_VAR
	VAR_INPUT
		nMaxLength	:	ULINT;	(* Maximum string length to export (including 0 termination). If the container content is longer, the string is cut off at nMaxLength - 1 and 0 termination is appended. In this case, S_FALSE is returned. *)
		hrPrev	:	HRESULT;	(* HRESULT indicating the result of previous operations (If SUCCEEDED(hrPrev) equals false, no operation is executed.) *)
	END_VAR

END_FUNCTION

// Functions/Basic Container Operations/F_VN_ExtractContainerRange

	{attribute 'TcIecLibraryType'}
	{attribute 'external_name' := 'F_VN_ExtractContainerRange_GUID_B64ED1A0_1B09_4861_EE07_7D23471534E2'}
	(* Copy the specified range of the source container into the destination container. (If the destination container already contains elements, they will be removed.) *)
	FUNCTION F_VN_ExtractContainerRange : HRESULT
	VAR_INPUT
		ipSrcContainer	:	ITcVnContainer;	(* Source container *)
		ipDestContainer	:	REFERENCE TO ITcVnContainer;	(* Destination container *)
		nFirstIdx	:	ULINT;	(* Index of the first element to copy *)
		nLastIdx	:	ULINT;	(* Index of the last element to copy *)
		hrPrev	:	HRESULT;	(* HRESULT indicating the result of previous operations (If SUCCEEDED(hrPrev) equals false, no operation is executed.) *)
	END_VAR

END_FUNCTION

// Functions/Basic Container Operations/F_VN_GetContainer

	{attribute 'TcIecLibraryType'}
	{attribute 'external_name' := 'F_VN_GetContainer_GUID_DFAC0E26_8EF4_4D8F_E803_980770171949'}
	(* Gets a pointer to the current element converted into an ITcVnContainer interface and increment its reference counter (only possible for container types). (Alternatively use interface method .GetContainer.) *)
	FUNCTION F_VN_GetContainer : HRESULT
	VAR_INPUT
		ipIterator	:	ITcVnForwardIterator;	(* Iterator *)
		ipContainer	:	REFERENCE TO ITcVnContainer;	(* Returns the container interface *)
		hrPrev	:	HRESULT;	(* HRESULT indicating the result of previous operations (If SUCCEEDED(hrPrev) equals false, no operation is executed.) *)
	END_VAR

END_FUNCTION

// Functions/Basic Container Operations/F_VN_GetContainerExp

	{attribute 'TcIecLibraryType'}
	{attribute 'external_name' := 'F_VN_GetContainerExp_GUID_BB90A4AB_E309_4D31_C2C3_93CADAB069A9'}
	(* Gets a pointer to the current element converted into an ITcVnContainer interface and increment its reference counter (only possible for container types). Additionally, an offset to increment or decrement the iterator afterwards can be provided. (expert function) *)
	FUNCTION F_VN_GetContainerExp : HRESULT
	VAR_INPUT
		ipIterator	:	ITcVnForwardIterator;	(* Iterator *)
		ipContainer	:	REFERENCE TO ITcVnContainer;	(* Returns the container interface *)
		nOffset	:	DINT;	(* Offset to increment (>0) or decrement (<0) the iterator afterwards *)
		hrPrev	:	HRESULT;	(* HRESULT indicating the result of previous operations (If SUCCEEDED(hrPrev) equals false, no operation is executed.) *)
	END_VAR

END_FUNCTION

// Functions/Basic Container Operations/F_VN_GetForwardIterator

	{attribute 'TcIecLibraryType'}
	{attribute 'external_name' := 'F_VN_GetForwardIterator_GUID_BBFBDA38_47EB_4B91_FB9F_A04484427AE0'}
	(* Gets a forward iterator for the container. (Alternatively use interface method .GetForwardIterator.) *)
	FUNCTION F_VN_GetForwardIterator : HRESULT
	VAR_INPUT
		ipContainer	:	ITcVnContainer;	(* Container *)
		ipIterator	:	REFERENCE TO ITcVnForwardIterator;	(* Returns the iterator interface *)
		hrPrev	:	HRESULT;	(* HRESULT indicating the result of previous operations (If SUCCEEDED(hrPrev) equals false, no operation is executed.) *)
	END_VAR

END_FUNCTION

// Functions/Basic Container Operations/F_VN_GetNumberOfElements

	{attribute 'TcIecLibraryType'}
	{attribute 'external_name' := 'F_VN_GetNumberOfElements_GUID_39941F40_DB03_4C2D_C898_22CF50A747AB'}
	(* Gets the number of elements in the container. (Alternatively use interface method .getElementNum.) *)
	FUNCTION F_VN_GetNumberOfElements : HRESULT
	VAR_INPUT
		ipContainer	:	ITcVnContainer;	(* Container *)
	END_VAR
	VAR_IN_OUT
		nNumberOfElements	:	ULINT;	(* Returns the number of elements in ipContainer *)
	END_VAR
	VAR_INPUT
		hrPrev	:	HRESULT;	(* HRESULT indicating the result of previous operations (If SUCCEEDED(hrPrev) equals false, no operation is executed.) *)
	END_VAR

END_FUNCTION

// Functions/Basic Container Operations/F_VN_GetRandomAccessIterator

	{attribute 'TcIecLibraryType'}
	{attribute 'external_name' := 'F_VN_GetRandomAccessIterator_GUID_C7557608_77B2_46C8_CD19_3EFF37F1B2E5'}
	(* Gets a random access iterator for the container. (Alternatively use interface method .GetRandomAccessIterator.) *)
	FUNCTION F_VN_GetRandomAccessIterator : HRESULT
	VAR_INPUT
		ipContainer	:	ITcVnContainer;	(* Container *)
		ipIterator	:	REFERENCE TO ITcVnRandomAccessIterator;	(* Returns the iterator interface *)
		hrPrev	:	HRESULT;	(* HRESULT indicating the result of previous operations (If SUCCEEDED(hrPrev) equals false, no operation is executed.) *)
	END_VAR

END_FUNCTION

// Functions/Basic Container Operations/F_VN_IncrementIterator

	{attribute 'TcIecLibraryType'}
	{attribute 'external_name' := 'F_VN_IncrementIterator_GUID_915D3FEE_4F0F_406C_DD1E_8104BF3CA1E6'}
	(* Increment the iterator. (Alternatively use interface method .Increment.) *)
	FUNCTION F_VN_IncrementIterator : HRESULT
	VAR_INPUT
		ipIterator	:	ITcVnForwardIterator;	(* Iterator *)
		hrPrev	:	HRESULT;	(* HRESULT indicating the result of previous operations (If SUCCEEDED(hrPrev) equals false, no operation is executed.) *)
	END_VAR

END_FUNCTION

// Functions/Basic Container Operations/F_VN_IteratorDistance

	{attribute 'TcIecLibraryType'}
	{attribute 'external_name' := 'F_VN_IteratorDistance_GUID_24EC6C63_693F_4237_E217_C5F9C9786870'}
	(* Computes the distance between 2 iterators. *)
	FUNCTION F_VN_IteratorDistance : HRESULT
	VAR_INPUT
		ipIteratorFirst	:	ITcVnForwardIterator;	(* First iterator *)
		ipIteratorLast	:	ITcVnForwardIterator;	(* Last iterator *)
	END_VAR
	VAR_IN_OUT
		nDistance	:	LINT;	(* Returns the computed distance *)
	END_VAR
	VAR_INPUT
		hrPrev	:	HRESULT;	(* HRESULT indicating the result of previous operations (If SUCCEEDED(hrPrev) equals false, no operation is executed.) *)
	END_VAR

END_FUNCTION

// Functions/Basic Container Operations/F_VN_ReserveContainerMemory

	{attribute 'TcIecLibraryType'}
	{attribute 'external_name' := 'F_VN_ReserveContainerMemory_GUID_5E35375E_4ACB_43F3_D0FA_772DD1DFC9DE'}
	(* Reserve container memory (call with maximum required number of elements before manually appending elements for better performance) *)
	FUNCTION F_VN_ReserveContainerMemory : HRESULT
	VAR_INPUT
		ipContainer	:	ITcVnContainer;	(* Container for which to reserve the memory *)
		nElements	:	ULINT;	(* Number of elements for which the container should reserve memory *)
		hrPrev	:	HRESULT;	(* HRESULT indicating the result of previous operations (If SUCCEEDED(hrPrev) equals false, no operation is executed.) *)
	END_VAR

END_FUNCTION

// Functions/Basic Container Operations/F_VN_ReverseContainer

	{attribute 'TcIecLibraryType'}
	{attribute 'external_name' := 'F_VN_ReverseContainer_GUID_CD0D47AD_2827_4E67_E6B3_FA30C11F3F50'}
	(* Reverse the container elements. *)
	FUNCTION F_VN_ReverseContainer : HRESULT
	VAR_INPUT
		ipContainer	:	ITcVnContainer;	(* Container to be reversed *)
		hrPrev	:	HRESULT;	(* HRESULT indicating the result of previous operations (If SUCCEEDED(hrPrev) equals false, no operation is executed.) *)
	END_VAR

END_FUNCTION

// Functions/Basic Container Operations/F_VN_SetContainer

	{attribute 'TcIecLibraryType'}
	{attribute 'external_name' := 'F_VN_SetContainer_GUID_1B6F2F6D_C5D6_4C49_C488_CE9ABEC6E050'}
	(* Sets the current element using an ITcVnContainer interface (only possible for container types). (Alternatively use interface method .SetContainer.) *)
	FUNCTION F_VN_SetContainer : HRESULT
	VAR_INPUT
		ipIterator	:	ITcVnForwardIterator;	(* Iterator *)
		ipContainer	:	ITcVnContainer;	(* Container interface of which the content is to be assigned to the current element *)
		hrPrev	:	HRESULT;	(* HRESULT indicating the result of previous operations (If SUCCEEDED(hrPrev) equals false, no operation is executed.) *)
	END_VAR

END_FUNCTION

// Functions/Basic Container Operations/F_VN_SetIteratorToBegin

	{attribute 'TcIecLibraryType'}
	{attribute 'external_name' := 'F_VN_SetIteratorToBegin_GUID_A9188DC1_FE4D_4021_F70A_2EC40588FEB8'}
	(* Sets the iterator to the first element of the container. (Alternatively use interface method .SetToBegin.) *)
	FUNCTION F_VN_SetIteratorToBegin : HRESULT
	VAR_INPUT
		ipIterator	:	ITcVnForwardIterator;	(* Iterator *)
		hrPrev	:	HRESULT;	(* HRESULT indicating the result of previous operations (If SUCCEEDED(hrPrev) equals false, no operation is executed.) *)
	END_VAR

END_FUNCTION

// Functions/Geometric and Coordinate Transformations/F_VN_AlignRotatedImageRegion

	{attribute 'TcIecLibraryType'}
	{attribute 'external_name' := 'F_VN_AlignRotatedImageRegion_GUID_C7DA0AA2_AE94_44AD_F466_E16EC44A8F52'}
	(* Copies the provided image region and aligns it to the image axes. *)
	FUNCTION F_VN_AlignRotatedImageRegion : HRESULT
	VAR_INPUT
		ipSrcImage	:	ITcVnImage;	(* Source image *)
		ipDestImage	:	REFERENCE TO ITcVnImage;	(* Destination image (An appropriate image will be created if required.) *)
	END_VAR
	VAR_IN_OUT
		stRegion	:	TcVnRotatedRectangle;	(* Image region to be aligned *)
	END_VAR
	VAR_INPUT
		hrPrev	:	HRESULT;	(* HRESULT indicating the result of previous operations (If SUCCEEDED(hrPrev) equals false, no operation is executed.) *)
	END_VAR

END_FUNCTION

// Functions/Geometric and Coordinate Transformations/F_VN_AlignRotatedImageRegionExp

	{attribute 'TcIecLibraryType'}
	{attribute 'external_name' := 'F_VN_AlignRotatedImageRegionExp_GUID_2BC60D0B_3156_4586_DD75_9F1ECFDD8842'}
	(* Copies the provided image region and aligns it to the image axes. (expert function) *)
	FUNCTION F_VN_AlignRotatedImageRegionExp : HRESULT
	VAR_INPUT
		ipSrcImage	:	ITcVnImage;	(* Source image *)
		ipDestImage	:	REFERENCE TO ITcVnImage;	(* Destination image (An appropriate image will be created if required.) *)
	END_VAR
	VAR_IN_OUT
		stRegion	:	TcVnRotatedRectangle;	(* Image region to be aligned *)
	END_VAR
	VAR_INPUT
		eInterpolationType	:	ETcVnInterpolationType;	(* Interpolation method *)
		eBorderInterpolation	:	ETcVnBorderInterpolationMethod;	(* Border interpolation method (ISOLATED not supported) *)
	END_VAR
	VAR_IN_OUT
		aBorderValue	:	TcVnVector4_LREAL;	(* Border value, if CONSTANT is used *)
	END_VAR
	VAR_INPUT
		hrPrev	:	HRESULT;	(* HRESULT indicating the result of previous operations (If SUCCEEDED(hrPrev) equals false, no operation is executed.) *)
	END_VAR

END_FUNCTION

// Functions/Geometric and Coordinate Transformations/F_VN_ApplyRotationToAffineTransformation

	{attribute 'TcIecLibraryType'}
	{attribute 'external_name' := 'F_VN_ApplyRotationToAffineTransformation_GUID_2A56BF14_D589_48A4_D443_095C0247BC71'}
	(* Apply a rotation to an existing 2D affine transformation matrix. *)
	FUNCTION F_VN_ApplyRotationToAffineTransformation : HRESULT
	VAR_IN_OUT
		aTransformationMatrix	:	TcVnMatrix2x3_LREAL;	(* Affine transformation matrix to which the rotation is applied *)
	END_VAR
	VAR_INPUT
		fAngle	:	LREAL;	(* Angle in radians (positive means counter-clockwise) *)
		hrPrev	:	HRESULT;	(* HRESULT indicating the result of previous operations (If SUCCEEDED(hrPrev) equals false, no operation is executed.) *)
	END_VAR

END_FUNCTION

// Functions/Geometric and Coordinate Transformations/F_VN_ApplyRotationToAffineTransformationExp

	{attribute 'TcIecLibraryType'}
	{attribute 'external_name' := 'F_VN_ApplyRotationToAffineTransformationExp_GUID_F17D445B_938B_4A47_C7C3_FA5F94E72629'}
	(* Apply a rotation to an existing 2D affine transformation matrix. (expert function) *)
	FUNCTION F_VN_ApplyRotationToAffineTransformationExp : HRESULT
	VAR_IN_OUT
		aTransformationMatrix	:	TcVnMatrix2x3_LREAL;	(* Affine transformation matrix to which the rotation is applied *)
	END_VAR
	VAR_INPUT
		fAngle	:	LREAL;	(* Angle in radians (positive means counter-clockwise) *)
		bUsePreMultiplication	:	BOOL;	(* Select if pre- or post-multiplication should be used *)
		hrPrev	:	HRESULT;	(* HRESULT indicating the result of previous operations (If SUCCEEDED(hrPrev) equals false, no operation is executed.) *)
	END_VAR

END_FUNCTION

// Functions/Geometric and Coordinate Transformations/F_VN_ApplyScalingToAffineTransformation

	{attribute 'TcIecLibraryType'}
	{attribute 'external_name' := 'F_VN_ApplyScalingToAffineTransformation_GUID_F23F2249_19C7_4DCB_C4E6_82E563385F76'}
	(* Apply a scaling to an existing 2D affine transformation matrix. *)
	FUNCTION F_VN_ApplyScalingToAffineTransformation : HRESULT
	VAR_IN_OUT
		aTransformationMatrix	:	TcVnMatrix2x3_LREAL;	(* Affine transformation matrix to which the scaling is applied *)
	END_VAR
	VAR_INPUT
		fScaleX	:	LREAL;	(* Scaling factor in x direction *)
		fScaleY	:	LREAL;	(* Scaling factor in y direction *)
		hrPrev	:	HRESULT;	(* HRESULT indicating the result of previous operations (If SUCCEEDED(hrPrev) equals false, no operation is executed.) *)
	END_VAR

END_FUNCTION

// Functions/Geometric and Coordinate Transformations/F_VN_ApplyScalingToAffineTransformationExp

	{attribute 'TcIecLibraryType'}
	{attribute 'external_name' := 'F_VN_ApplyScalingToAffineTransformationExp_GUID_F3E198C6_7077_469B_F934_DF77865294DF'}
	(* Apply a scaling to an existing 2D affine transformation matrix. (expert function) *)
	FUNCTION F_VN_ApplyScalingToAffineTransformationExp : HRESULT
	VAR_IN_OUT
		aTransformationMatrix	:	TcVnMatrix2x3_LREAL;	(* Affine transformation matrix to which the scaling is applied *)
	END_VAR
	VAR_INPUT
		fScaleX	:	LREAL;	(* Scaling factor in x direction *)
		fScaleY	:	LREAL;	(* Scaling factor in y direction *)
		bUsePreMultiplication	:	BOOL;	(* Select if pre- or post-multiplication should be used *)
		hrPrev	:	HRESULT;	(* HRESULT indicating the result of previous operations (If SUCCEEDED(hrPrev) equals false, no operation is executed.) *)
	END_VAR

END_FUNCTION

// Functions/Geometric and Coordinate Transformations/F_VN_ApplyTranslationToAffineTransformation

	{attribute 'TcIecLibraryType'}
	{attribute 'external_name' := 'F_VN_ApplyTranslationToAffineTransformation_GUID_D41F639E_9FAC_43BB_C019_2F72A960205E'}
	(* Apply a translation to an existing 2D affine transformation matrix. *)
	FUNCTION F_VN_ApplyTranslationToAffineTransformation : HRESULT
	VAR_IN_OUT
		aTransformationMatrix	:	TcVnMatrix2x3_LREAL;	(* Affine transformation matrix to which the translation is applied *)
	END_VAR
	VAR_INPUT
		fDeltaX	:	LREAL;	(* Translation in x direction *)
		fDeltaY	:	LREAL;	(* Translation in y direction *)
		hrPrev	:	HRESULT;	(* HRESULT indicating the result of previous operations (If SUCCEEDED(hrPrev) equals false, no operation is executed.) *)
	END_VAR

END_FUNCTION

// Functions/Geometric and Coordinate Transformations/F_VN_ApplyTranslationToAffineTransformationExp

	{attribute 'TcIecLibraryType'}
	{attribute 'external_name' := 'F_VN_ApplyTranslationToAffineTransformationExp_GUID_4C725624_EF2A_4897_C84A_7763D2C1096B'}
	(* Apply a translation to an existing 2D affine transformation matrix. (expert function) *)
	FUNCTION F_VN_ApplyTranslationToAffineTransformationExp : HRESULT
	VAR_IN_OUT
		aTransformationMatrix	:	TcVnMatrix2x3_LREAL;	(* Affine transformation matrix to which the translation is applied *)
	END_VAR
	VAR_INPUT
		fDeltaX	:	LREAL;	(* Translation in x direction *)
		fDeltaY	:	LREAL;	(* Translation in y direction *)
		bUsePreMultiplication	:	BOOL;	(* Select if pre- or post-multiplication should be used *)
		hrPrev	:	HRESULT;	(* HRESULT indicating the result of previous operations (If SUCCEEDED(hrPrev) equals false, no operation is executed.) *)
	END_VAR

END_FUNCTION

// Functions/Geometric and Coordinate Transformations/F_VN_ApplyYAxisInversionToAffineTransformation

	{attribute 'TcIecLibraryType'}
	{attribute 'external_name' := 'F_VN_ApplyYAxisInversionToAffineTransformation_GUID_535BEC6A_1EDF_4B25_F635_8F95A99AEFF1'}
	(* Apply an inversion of the y-axis direction to an existing 2D affine transformation matrix. *)
	FUNCTION F_VN_ApplyYAxisInversionToAffineTransformation : HRESULT
	VAR_IN_OUT
		aTransformationMatrix	:	TcVnMatrix2x3_LREAL;	(* Affine transformation matrix to which the inversion of the y-axis direction is applied *)
	END_VAR
	VAR_INPUT
		hrPrev	:	HRESULT;	(* HRESULT indicating the result of previous operations (If SUCCEEDED(hrPrev) equals false, no operation is executed.) *)
	END_VAR

END_FUNCTION

// Functions/Geometric and Coordinate Transformations/F_VN_ApplyYAxisInversionToAffineTransformationExp

	{attribute 'TcIecLibraryType'}
	{attribute 'external_name' := 'F_VN_ApplyYAxisInversionToAffineTransformationExp_GUID_FDE560C4_3F3C_46CF_D00F_7F53477D4BF6'}
	(* Apply an inversion of the y-axis direction to an existing 2D affine transformation matrix. (expert function) *)
	FUNCTION F_VN_ApplyYAxisInversionToAffineTransformationExp : HRESULT
	VAR_IN_OUT
		aTransformationMatrix	:	TcVnMatrix2x3_LREAL;	(* Affine transformation matrix to which the inversion of the y-axis direction is applied *)
	END_VAR
	VAR_INPUT
		bUsePreMultiplication	:	BOOL;	(* Select if pre- or post-multiplication should be used *)
		hrPrev	:	HRESULT;	(* HRESULT indicating the result of previous operations (If SUCCEEDED(hrPrev) equals false, no operation is executed.) *)
	END_VAR

END_FUNCTION

// Functions/Geometric and Coordinate Transformations/F_VN_ConvertCartesianToPolarAngleImage

	{attribute 'TcIecLibraryType'}
	{attribute 'external_name' := 'F_VN_ConvertCartesianToPolarAngleImage_GUID_EF168EF5_E538_42ED_EF95_C80A6DA04CF6'}
	(* Converts cartesian coordinates (x, y) to polar angle. *)
	FUNCTION F_VN_ConvertCartesianToPolarAngleImage : HRESULT
	VAR_INPUT
		ipSrcImageX	:	ITcVnImage;	(* Source image containing the x values (elements of type REAL or LREAL) *)
		ipSrcImageY	:	ITcVnImage;	(* Source image containing the y values (Same element type as ipSrcImageX) *)
		ipDestImageAng	:	REFERENCE TO ITcVnImage;	(* Destination image containing the angles (Same element type as source images. An appropriate destination image will be created if required.) *)
		hrPrev	:	HRESULT;	(* HRESULT indicating the result of previous operations (If SUCCEEDED(hrPrev) equals false, no operation is executed.) *)
	END_VAR

END_FUNCTION

// Functions/Geometric and Coordinate Transformations/F_VN_ConvertCartesianToPolarAngleImageExp

	{attribute 'TcIecLibraryType'}
	{attribute 'external_name' := 'F_VN_ConvertCartesianToPolarAngleImageExp_GUID_E5942133_3AB5_473A_EBCD_EE7EBFCA686D'}
	(* Converts cartesian coordinates (x, y) to polar angle. (expert function) *)
	FUNCTION F_VN_ConvertCartesianToPolarAngleImageExp : HRESULT
	VAR_INPUT
		ipSrcImageX	:	ITcVnImage;	(* Source image containing the x values (elements of type REAL or LREAL) *)
		ipSrcImageY	:	ITcVnImage;	(* Source image containing the y values (Same element type as ipSrcImageX) *)
		ipDestImageAng	:	REFERENCE TO ITcVnImage;	(* Destination image containing the angles (Same element type as source images. An appropriate destination image will be created if required.) *)
		bAngleInDegrees	:	BOOL;	(* Specifys, if the angles should be in degrees or radians *)
		hrPrev	:	HRESULT;	(* HRESULT indicating the result of previous operations (If SUCCEEDED(hrPrev) equals false, no operation is executed.) *)
	END_VAR

END_FUNCTION

// Functions/Geometric and Coordinate Transformations/F_VN_ConvertCartesianToPolarAngles

	{attribute 'TcIecLibraryType'}
	{attribute 'external_name' := 'F_VN_ConvertCartesianToPolarAngles_GUID_1FE81EFF_0370_43A0_D77F_274AB43D7DAC'}
	(* Converts cartesian coordinates (x, y) to polar angle. *)
	FUNCTION F_VN_ConvertCartesianToPolarAngles : HRESULT
	VAR_INPUT
		ipSrcPointsCart	:	ITcVnContainer;	(* Container with cartesian points (ContainerType_Vector_TcVnPoint2_DINT or ContainerType_Vector_TcVnPoint2_REAL or ContainerType_Vector_TcVnPoint2_LREAL) *)
		ipDestAngles	:	REFERENCE TO ITcVnContainer;	(* Returns a container which is filled with the angles (ContainerType_Vector_REAL, if source points are of type TcVnPoint2_DINT or TcVnPoint2_REAL; else ContainerType_Vector_LREAL. Non-zero interface pointers are reused.) *)
		hrPrev	:	HRESULT;	(* HRESULT indicating the result of previous operations (If SUCCEEDED(hrPrev) equals false, no operation is executed.) *)
	END_VAR

END_FUNCTION

// Functions/Geometric and Coordinate Transformations/F_VN_ConvertCartesianToPolarAnglesExp

	{attribute 'TcIecLibraryType'}
	{attribute 'external_name' := 'F_VN_ConvertCartesianToPolarAnglesExp_GUID_A9E8EDF6_CDA0_44A3_D480_F77BE45FDCC9'}
	(* Converts cartesian coordinates (x, y) to polar angle. (expert function) *)
	FUNCTION F_VN_ConvertCartesianToPolarAnglesExp : HRESULT
	VAR_INPUT
		ipSrcPointsCart	:	ITcVnContainer;	(* Container with cartesian points (ContainerType_Vector_TcVnPoint2_DINT or ContainerType_Vector_TcVnPoint2_REAL or ContainerType_Vector_TcVnPoint2_LREAL) *)
		ipDestAngles	:	REFERENCE TO ITcVnContainer;	(* Returns a container which is filled with the angles (ContainerType_Vector_REAL, if source points are of type TcVnPoint2_DINT or TcVnPoint2_REAL; else ContainerType_Vector_LREAL. Non-zero interface pointers are reused.) *)
		bAngleInDegrees	:	BOOL;	(* Specify, if the angles should be in degrees or radians *)
		hrPrev	:	HRESULT;	(* HRESULT indicating the result of previous operations (If SUCCEEDED(hrPrev) equals false, no operation is executed.) *)
	END_VAR

END_FUNCTION

// Functions/Geometric and Coordinate Transformations/F_VN_ConvertCartesianToPolarImages

	{attribute 'TcIecLibraryType'}
	{attribute 'external_name' := 'F_VN_ConvertCartesianToPolarImages_GUID_00465D3A_ACC9_45E7_E873_95BA43C8D3F2'}
	(* Converts cartesian coordinates (x, y) to polar coordinates (magnitude, angle). *)
	FUNCTION F_VN_ConvertCartesianToPolarImages : HRESULT
	VAR_INPUT
		ipSrcImageX	:	ITcVnImage;	(* Source image containing the x values (elements of type REAL or LREAL) *)
		ipSrcImageY	:	ITcVnImage;	(* Source image containing the y values (Same element type as ipSrcImageX) *)
		ipDestImageMag	:	REFERENCE TO ITcVnImage;	(* Destination image containing the magnitudes (Same element type as source images. An appropriate destination image will be created if required.) *)
		ipDestImageAng	:	REFERENCE TO ITcVnImage;	(* Destination image containing the angles (Same element type as source images. An appropriate destination image will be created if required.) *)
		hrPrev	:	HRESULT;	(* HRESULT indicating the result of previous operations (If SUCCEEDED(hrPrev) equals false, no operation is executed.) *)
	END_VAR

END_FUNCTION

// Functions/Geometric and Coordinate Transformations/F_VN_ConvertCartesianToPolarImagesExp

	{attribute 'TcIecLibraryType'}
	{attribute 'external_name' := 'F_VN_ConvertCartesianToPolarImagesExp_GUID_3F373B67_C7FD_4448_FF3B_582FBC5A4A3B'}
	(* Converts cartesian coordinates (x, y) to polar coordinates (magnitude, angle). (expert function) *)
	FUNCTION F_VN_ConvertCartesianToPolarImagesExp : HRESULT
	VAR_INPUT
		ipSrcImageX	:	ITcVnImage;	(* Source image containing the x values (elements of type REAL or LREAL) *)
		ipSrcImageY	:	ITcVnImage;	(* Source image containing the y values (Same element type as ipSrcImageX) *)
		ipDestImageMag	:	REFERENCE TO ITcVnImage;	(* Destination image containing the magnitudes (Same element type as source images. An appropriate destination image will be created if required.) *)
		ipDestImageAng	:	REFERENCE TO ITcVnImage;	(* Destination image containing the angles (Same element type as source images. An appropriate destination image will be created if required.) *)
		bAngleInDegrees	:	BOOL;	(* Specifys, if the angles should be in degrees or radians *)
		hrPrev	:	HRESULT;	(* HRESULT indicating the result of previous operations (If SUCCEEDED(hrPrev) equals false, no operation is executed.) *)
	END_VAR

END_FUNCTION

// Functions/Geometric and Coordinate Transformations/F_VN_ConvertCartesianToPolarMagnitudeImage

	{attribute 'TcIecLibraryType'}
	{attribute 'external_name' := 'F_VN_ConvertCartesianToPolarMagnitudeImage_GUID_F17C8165_A8B9_44A2_E824_99E66007458C'}
	(* Converts cartesian coordinates (x, y) to polar magnitude. *)
	FUNCTION F_VN_ConvertCartesianToPolarMagnitudeImage : HRESULT
	VAR_INPUT
		ipSrcImageX	:	ITcVnImage;	(* Source image containing the x values (elements of type REAL or LREAL) *)
		ipSrcImageY	:	ITcVnImage;	(* Source image containing the y values (Same element type as ipSrcImageX) *)
		ipDestImageMag	:	REFERENCE TO ITcVnImage;	(* Destination image containing the magnitudes (Same element type as source images. An appropriate destination image will be created if required.) *)
		hrPrev	:	HRESULT;	(* HRESULT indicating the result of previous operations (If SUCCEEDED(hrPrev) equals false, no operation is executed.) *)
	END_VAR

END_FUNCTION

// Functions/Geometric and Coordinate Transformations/F_VN_ConvertCartesianToPolarMagnitudes

	{attribute 'TcIecLibraryType'}
	{attribute 'external_name' := 'F_VN_ConvertCartesianToPolarMagnitudes_GUID_EFC402B7_5E34_4945_E6CB_E3CBD3B5D092'}
	(* Converts cartesian coordinates (x, y) to polar magnitude. *)
	FUNCTION F_VN_ConvertCartesianToPolarMagnitudes : HRESULT
	VAR_INPUT
		ipSrcPointsCart	:	ITcVnContainer;	(* Container with cartesian points (ContainerType_Vector_TcVnPoint2_DINT or ContainerType_Vector_TcVnPoint2_REAL or ContainerType_Vector_TcVnPoint2_LREAL) *)
		ipDestMags	:	REFERENCE TO ITcVnContainer;	(* Returns a container which is filled with the magnitudes (ContainerType_Vector_REAL, if source points are of type TcVnPoint2_DINT or TcVnPoint2_REAL; else ContainerType_Vector_LREAL. Non-zero interface pointers are reused.) *)
		hrPrev	:	HRESULT;	(* HRESULT indicating the result of previous operations (If SUCCEEDED(hrPrev) equals false, no operation is executed.) *)
	END_VAR

END_FUNCTION

// Functions/Geometric and Coordinate Transformations/F_VN_ConvertCartesianToPolarPoints

	{attribute 'TcIecLibraryType'}
	{attribute 'external_name' := 'F_VN_ConvertCartesianToPolarPoints_GUID_E382B624_23DF_4283_DEC6_0CAD68676736'}
	(* Converts cartesian coordinates (x, y) to polar coordinates (magnitude, angle). *)
	FUNCTION F_VN_ConvertCartesianToPolarPoints : HRESULT
	VAR_INPUT
		ipSrcPointsCart	:	ITcVnContainer;	(* Container with cartesian points (ContainerType_Vector_TcVnPoint2_DINT or ContainerType_Vector_TcVnPoint2_REAL or ContainerType_Vector_TcVnPoint2_LREAL) *)
		ipDestPointsPolar	:	REFERENCE TO ITcVnContainer;	(* Returns a container which is filled with the converted points in polar coordinates (ContainerType_Vector_TcVnPoint2_REAL, if source points are of type TcVnPoint2_DINT or TcVnPoint2_REAL; else ContainerType_Vector_TcVnPoint2_LREAL. Non-zero interface pointers are reused.) *)
		hrPrev	:	HRESULT;	(* HRESULT indicating the result of previous operations (If SUCCEEDED(hrPrev) equals false, no operation is executed.) *)
	END_VAR

END_FUNCTION

// Functions/Geometric and Coordinate Transformations/F_VN_ConvertCartesianToPolarPointsExp

	{attribute 'TcIecLibraryType'}
	{attribute 'external_name' := 'F_VN_ConvertCartesianToPolarPointsExp_GUID_832D10CF_4569_4F1B_FF14_4307BB2D3517'}
	(* Converts cartesian coordinates (x, y) to polar coordinates (magnitude, angle). (expert function) *)
	FUNCTION F_VN_ConvertCartesianToPolarPointsExp : HRESULT
	VAR_INPUT
		ipSrcPointsCart	:	ITcVnContainer;	(* Container with cartesian points (ContainerType_Vector_TcVnPoint2_DINT or ContainerType_Vector_TcVnPoint2_REAL or ContainerType_Vector_TcVnPoint2_LREAL) *)
		ipDestPointsPolar	:	REFERENCE TO ITcVnContainer;	(* Returns a container which is filled with the converted points in polar coordinates (ContainerType_Vector_TcVnPoint2_REAL, if source points are of type TcVnPoint2_DINT or TcVnPoint2_REAL; else ContainerType_Vector_TcVnPoint2_LREAL. Non-zero interface pointers are reused.) *)
		bAngleInDegrees	:	BOOL;	(* Specifys, if the angles should be in degrees or radians *)
		hrPrev	:	HRESULT;	(* HRESULT indicating the result of previous operations (If SUCCEEDED(hrPrev) equals false, no operation is executed.) *)
	END_VAR

END_FUNCTION

// Functions/Geometric and Coordinate Transformations/F_VN_ConvertPolarToCartesianImages

	{attribute 'TcIecLibraryType'}
	{attribute 'external_name' := 'F_VN_ConvertPolarToCartesianImages_GUID_2D71C191_E682_410F_F4FB_41C6D577485A'}
	(* Converts polar coordinates (magnitude, angle) to cartesian coordinates (x, y). *)
	FUNCTION F_VN_ConvertPolarToCartesianImages : HRESULT
	VAR_INPUT
		ipSrcImageMag	:	ITcVnImage;	(* Source image containing the magnitudes (elements of type REAL or LREAL) *)
		ipSrcImageAng	:	ITcVnImage;	(* Source image containing the angles (Same element type as ipSrcImageMag) *)
		ipDestImageX	:	REFERENCE TO ITcVnImage;	(* Destination image containing the x values (Same element type as source images. An appropriate destination image will be created if required.) *)
		ipDestImageY	:	REFERENCE TO ITcVnImage;	(* Destination image containing the y values (Same element type as source images. An appropriate destination image will be created if required.) *)
		hrPrev	:	HRESULT;	(* HRESULT indicating the result of previous operations (If SUCCEEDED(hrPrev) equals false, no operation is executed.) *)
	END_VAR

END_FUNCTION

// Functions/Geometric and Coordinate Transformations/F_VN_ConvertPolarToCartesianImagesExp

	{attribute 'TcIecLibraryType'}
	{attribute 'external_name' := 'F_VN_ConvertPolarToCartesianImagesExp_GUID_722696ED_540C_4A30_C69D_F281806B2717'}
	(* Converts polar coordinates (magnitude, angle) to cartesian coordinates (x, y). (expert function) *)
	FUNCTION F_VN_ConvertPolarToCartesianImagesExp : HRESULT
	VAR_INPUT
		ipSrcImageMag	:	ITcVnImage;	(* Source image containing the magnitudes (elements of type REAL or LREAL) *)
		ipSrcImageAng	:	ITcVnImage;	(* Source image containing the angles (Same element type as ipSrcImageMag) *)
		ipDestImageX	:	REFERENCE TO ITcVnImage;	(* Destination image containing the x values (Same element type as source images. An appropriate destination image will be created if required.) *)
		ipDestImageY	:	REFERENCE TO ITcVnImage;	(* Destination image containing the y values (Same element type as source images. An appropriate destination image will be created if required.) *)
		bAngleInDegrees	:	BOOL;	(* Specifys, if the angles are in degrees or radians *)
		hrPrev	:	HRESULT;	(* HRESULT indicating the result of previous operations (If SUCCEEDED(hrPrev) equals false, no operation is executed.) *)
	END_VAR

END_FUNCTION

// Functions/Geometric and Coordinate Transformations/F_VN_ConvertPolarToCartesianPoints

	{attribute 'TcIecLibraryType'}
	{attribute 'external_name' := 'F_VN_ConvertPolarToCartesianPoints_GUID_A50A4EB4_DDFA_4B42_C3A3_04E96C8E7A0A'}
	(* Converts polar coordinates (magnitude, angle) to cartesian coordinates (x, y). *)
	FUNCTION F_VN_ConvertPolarToCartesianPoints : HRESULT
	VAR_INPUT
		ipSrcPointsPolar	:	ITcVnContainer;	(* Container with polar coordinates (ContainerType_Vector_TcVnPoint2_REAL or ContainerType_Vector_TcVnPoint2_LREAL) *)
		ipDestPointsCart	:	REFERENCE TO ITcVnContainer;	(* Returns a container which is filled with the converted points in cartesian coordinates (same type ID as ipSrcPointsPolar. Non-zero interface pointers are reused.) *)
		hrPrev	:	HRESULT;	(* HRESULT indicating the result of previous operations (If SUCCEEDED(hrPrev) equals false, no operation is executed.) *)
	END_VAR

END_FUNCTION

// Functions/Geometric and Coordinate Transformations/F_VN_ConvertPolarToCartesianPointsExp

	{attribute 'TcIecLibraryType'}
	{attribute 'external_name' := 'F_VN_ConvertPolarToCartesianPointsExp_GUID_F91C1183_E799_4A7F_C954_885C157571C3'}
	(* Converts polar coordinates (magnitude, angle) to cartesian coordinates (x, y). (expert function) *)
	FUNCTION F_VN_ConvertPolarToCartesianPointsExp : HRESULT
	VAR_INPUT
		ipSrcPointsPolar	:	ITcVnContainer;	(* Container with polar coordinates (ContainerType_Vector_TcVnPoint2_REAL or ContainerType_Vector_TcVnPoint2_LREAL) *)
		ipDestPointsCart	:	REFERENCE TO ITcVnContainer;	(* Returns a container which is filled with the converted points in cartesian coordinates (same type ID as ipSrcPointsPolar. Non-zero interface pointers are reused.) *)
		bAngleInDegrees	:	BOOL;	(* Specifys, if the angles are in degrees or radians *)
		hrPrev	:	HRESULT;	(* HRESULT indicating the result of previous operations (If SUCCEEDED(hrPrev) equals false, no operation is executed.) *)
	END_VAR

END_FUNCTION

// Functions/Geometric and Coordinate Transformations/F_VN_DecomposeAffineTransformation

	{attribute 'TcIecLibraryType'}
	{attribute 'external_name' := 'F_VN_DecomposeAffineTransformation_GUID_F04692E7_E175_44F6_C3E5_C9F17C37DFB1'}
	(* Decompose an affine transformation matrix and return the rotation angle (clockwise) in radian. The decomposition method assumes the following order of transformation: Translation, Rotation, Scale, and Skew. *)
	FUNCTION F_VN_DecomposeAffineTransformation : HRESULT
	VAR_IN_OUT
		aAffineTransform	:	TcVnMatrix2x3_LREAL;	(* Affine transformation matrix *)
		fRotationAngle	:	LREAL;	(* Rotation angle (radian) in the clockwise direction. The rotation center is the origin point (0,0) *)
	END_VAR
	VAR_INPUT
		hrPrev	:	HRESULT;	(* HRESULT indicating the result of previous operations (If SUCCEEDED(hrPrev) equals false, no operation is executed.) *)
	END_VAR

END_FUNCTION

// Functions/Geometric and Coordinate Transformations/F_VN_DecomposeAffineTransformationExp

	{attribute 'TcIecLibraryType'}
	{attribute 'external_name' := 'F_VN_DecomposeAffineTransformationExp_GUID_F2E5EE7B_F870_4875_EE66_1AA4487B6A20'}
	(* Decompose an affine transformation matrix and return the rotation angle (clockwise) in radian, translation vector (pixels), scale, and skew vectors (angle in radian). The decomposition method assumes the following order of transformation: Translation, Rotation, Scale, and Skew. *)
	FUNCTION F_VN_DecomposeAffineTransformationExp : HRESULT
	VAR_IN_OUT
		aAffineTransform	:	TcVnMatrix2x3_LREAL;	(* Affine transformation matrix *)
		fRotationAngle	:	LREAL;	(* Rotation angle (radian) in the clockwise direction. The rotation center is the origin point (0,0) *)
		aTranslationVector	:	TcVnVector2_LREAL;	(* 2D translation vector. The values are in pixels *)
		aScaleVector	:	TcVnVector2_LREAL;	(* 2D scale vector  *)
		aSkewVector	:	TcVnVector2_LREAL;	(* 2D skew vector. The values are the skew angles in x and y directions in radian *)
	END_VAR
	VAR_INPUT
		hrPrev	:	HRESULT;	(* HRESULT indicating the result of previous operations (If SUCCEEDED(hrPrev) equals false, no operation is executed.) *)
	END_VAR

END_FUNCTION

// Functions/Geometric and Coordinate Transformations/F_VN_DecomposeHomography

	{attribute 'TcIecLibraryType'}
	{attribute 'external_name' := 'F_VN_DecomposeHomography_GUID_F0634BEF_7A15_488E_EDA1_BF7D6C46B892'}
	(* Decompose a homography matrix into four solutions of rotation, translation, and plane normal. It returns two solutions (Ra, Ta, Nb) and (Rb, Tb, Nb). The third and the fourth solutions can be calculated as follows: (Ra, -Ta, -Na) and (Rb, -Tb, -Nb). *)
	FUNCTION F_VN_DecomposeHomography : HRESULT
	VAR_IN_OUT
		aHomography	:	TcVnMatrix3x3_LREAL;	(* Homography matrix (a perspective transformation between two planes) *)
		aCameraMatrix	:	TcVnMatrix3x3_LREAL;	(* Camera matrix *)
		aRotationMatrixA	:	TcVnMatrix3x3_LREAL;	(* Rotation matrix of the first solution (Ra) *)
		aTranslationVectorA	:	TcVnVector3_LREAL;	(* Translation vector of the first solution (Ta) *)
		aNormVectorA	:	TcVnVector3_LREAL;	(* Norm vector of the first solution (Na) *)
		aRotationMatrixB	:	TcVnMatrix3x3_LREAL;	(* Rotation matrix of the second solution (Rb) *)
		aTranslationVectorB	:	TcVnVector3_LREAL;	(* Translation vector of the second solution (Tb) *)
		aNormVectorB	:	TcVnVector3_LREAL;	(* Norm vector of the second solution Nb *)
	END_VAR
	VAR_INPUT
		hrPrev	:	HRESULT;	(* HRESULT indicating the result of previous operations (If SUCCEEDED(hrPrev) equals false, no operation is executed.) *)
	END_VAR
	VAR_OUTPUT
		nSolutions	:	UDINT;	(* Returns the number of solutions. In normal cases, it is equal four.  *)
	END_VAR

END_FUNCTION

// Functions/Geometric and Coordinate Transformations/F_VN_DecomposeHomographyExp

	{attribute 'TcIecLibraryType'}
	{attribute 'external_name' := 'F_VN_DecomposeHomographyExp_GUID_8CC01627_964D_448A_ECF5_5CA72C24213C'}
	(* Decompose a homography matrix and verify four solutions of rotation, translation, and plane normal. It uses visible reference points being in front of the camera to confirm which solution(s) of the four solutions (maximum two solutions) are consistent with all reference points. *)
	FUNCTION F_VN_DecomposeHomographyExp : HRESULT
	VAR_IN_OUT
		aHomography	:	TcVnMatrix3x3_LREAL;	(* Homography matrix (a perspective transformation between two planes) *)
		aCameraMatrix	:	TcVnMatrix3x3_LREAL;	(* Camera matrix *)
		aRotationMatrixA	:	TcVnMatrix3x3_LREAL;	(* Rotation matrix of the first solution (Ra) *)
		aTranslationVectorA	:	TcVnVector3_LREAL;	(* Translation vector of the first solution (Ta) *)
		aNormVectorA	:	TcVnVector3_LREAL;	(* Norm vector of the first solution (Na) *)
		aRotationMatrixB	:	TcVnMatrix3x3_LREAL;	(* Rotation matrix of the second solution (Rb) *)
		aTranslationVectorB	:	TcVnVector3_LREAL;	(* Translation vector of the second solution (Tb) *)
		aNormVectorB	:	TcVnVector3_LREAL;	(* Norm vector of the second solution (Nb) *)
	END_VAR
	VAR_INPUT
		ipPointsSrc	:	ITcVnContainer;	(* Container with source points (ContainerType_Vector_TcVnPoint2_REAL) *)
		ipPointsDes	:	ITcVnContainer;	(* Container with destination points (same number as ipPoints1, ContainerType_Vector_TcVnPoint2_REAL) *)
		ipInlierMask	:	ITcVnContainer;	(* A mask marking the inliers (optional, set to 0 if not available; ContainerType_Vector_SINT or ContainerType_Vector_USINT) *)
		hrPrev	:	HRESULT;	(* HRESULT indicating the result of previous operations (If SUCCEEDED(hrPrev) equals false, no operation is executed.) *)
	END_VAR
	VAR_OUTPUT
		nSolutions	:	UDINT;	(* Return the number of true potential solutions [0,1, or 2].
							0: no true potential solutions for the given corresponding points are confirmed.
							1: the solution (Ra, Ta, Na) is confirmed.
							2: both solution (Ra, Ta, Na) and (Rb, Tb, Nb) are confirmed.
							In all cases the function returns two solutions (Ra, Ta, Nb) and (Rb, Tb, Nb). The third and the fourth solutions can be calculated as follows: (Ra, -Ta, -Na) and (Rb, -Tb, -Nb).
						 *)
	END_VAR

END_FUNCTION

// Functions/Geometric and Coordinate Transformations/F_VN_FlipImage

	{attribute 'TcIecLibraryType'}
	{attribute 'external_name' := 'F_VN_FlipImage_GUID_20207FD7_0167_4CB0_ED6A_989573BED795'}
	(* Flip an image (mirror and shift back to prior coordinates). *)
	FUNCTION F_VN_FlipImage : HRESULT
	VAR_INPUT
		ipSrcImage	:	ITcVnImage;	(* Source image *)
		ipDestImage	:	REFERENCE TO ITcVnImage;	(* Destination image (An appropriate destination image will be created if required.) *)
		eFlipAxis	:	ETcVnFlipAxis;	(* Selects the axis around which to flip the image *)
		hrPrev	:	HRESULT;	(* HRESULT indicating the result of previous operations (If SUCCEEDED(hrPrev) equals false, no operation is executed.) *)
	END_VAR

END_FUNCTION

// Functions/Geometric and Coordinate Transformations/F_VN_GenerateAffineTransformationUnitMatrix2D

	{attribute 'TcIecLibraryType'}
	{attribute 'external_name' := 'F_VN_GenerateAffineTransformationUnitMatrix2D_GUID_66E531E2_227B_4281_EA1C_090EA154798F'}
	(* Generate an affine transformation 2D unit matrix. *)
	FUNCTION F_VN_GenerateAffineTransformationUnitMatrix2D : HRESULT
	VAR_IN_OUT
		aTransformationMatrix	:	TcVnMatrix2x3_LREAL;	(* Resulting affine transformation unit matrix *)
	END_VAR
	VAR_INPUT
		hrPrev	:	HRESULT;	(* HRESULT indicating the result of previous operations (If SUCCEEDED(hrPrev) equals false, no operation is executed.) *)
	END_VAR

END_FUNCTION

// Functions/Geometric and Coordinate Transformations/F_VN_GetAffineTransformation

	{attribute 'TcIecLibraryType'}
	{attribute 'external_name' := 'F_VN_GetAffineTransformation_GUID_17072409_A76E_462E_EE6D_A310020B6523'}
	(* Calculate the affine transformation between three corresponding point pairs. The points mark the corners of the corresponding triangles. *)
	FUNCTION F_VN_GetAffineTransformation : HRESULT
	VAR_IN_OUT
		aSrcPoints	:	TcVnArray3_Point2_REAL;	(* Source points *)
		aDestPoints	:	TcVnArray3_Point2_REAL;	(* Destination points *)
		aTransformationMatrix	:	TcVnMatrix2x3_LREAL;	(* Resulting transformation matrix *)
	END_VAR
	VAR_INPUT
		hrPrev	:	HRESULT;	(* HRESULT indicating the result of previous operations (If SUCCEEDED(hrPrev) equals false, no operation is executed.) *)
	END_VAR

END_FUNCTION

// Functions/Geometric and Coordinate Transformations/F_VN_GetAffineTransformation2D

	{attribute 'TcIecLibraryType'}
	{attribute 'external_name' := 'F_VN_GetAffineTransformation2D_GUID_1D5CE630_28BD_4FBA_E030_06B2B5DEEB3F'}
	(* Estimate the 2D affine transformation between two planar point sets using RANSAC algorithm. *)
	FUNCTION F_VN_GetAffineTransformation2D : HRESULT
	VAR_INPUT
		ipSrcPoints	:	ITcVnContainer;	(* Container with at least 3 source points (ContainerType_Vector_TcVnPoint2_REAL) *)
		ipDestPoints	:	ITcVnContainer;	(* Container with destination points (same number as ipSrcPoints, ContainerType_Vector_TcVnPoint2_REAL) *)
	END_VAR
	VAR_IN_OUT
		aAffineTransform	:	TcVnMatrix2x3_LREAL;	(* Returns the affine transformation matrix, which transforms the source points to the destination points *)
	END_VAR
	VAR_INPUT
		hrPrev	:	HRESULT;	(* HRESULT indicating the result of previous operations (If SUCCEEDED(hrPrev) equals false, no operation is executed.) *)
	END_VAR

END_FUNCTION

// Functions/Geometric and Coordinate Transformations/F_VN_GetAffineTransformation2DExp

	{attribute 'TcIecLibraryType'}
	{attribute 'external_name' := 'F_VN_GetAffineTransformation2DExp_GUID_CFBDE160_2378_4CA5_EE23_F380F58634BC'}
	(* Estimate the affine transformation between two planar point sets. (expert function) *)
	FUNCTION F_VN_GetAffineTransformation2DExp : HRESULT
	VAR_INPUT
		ipSrcPoints	:	ITcVnContainer;	(* Container with at least 3 source points (ContainerType_Vector_TcVnPoint2_REAL) *)
		ipDestPoints	:	ITcVnContainer;	(* Container with destination points (same number as ipSrcPoints, ContainerType_Vector_TcVnPoint2_REAL) *)
	END_VAR
	VAR_IN_OUT
		aAffineTransform	:	TcVnMatrix2x3_LREAL;	(* Returns the affine transformation matrix, which transforms the source points to the destination points *)
	END_VAR
	VAR_INPUT
		eAlgorithm	:	ETcVnEstimationAlgorithm;	(* Estimation algorithm (only RANSAC and LMEDS are supported) *)
		fReprojThreshold	:	LREAL;	(* Maximum allowed reprojection error to treat a point pair as an inlier *)
		ipInlierMask	:	REFERENCE TO ITcVnContainer;	(* Returns a mask marking the inliers (optional, set to 0 if not required; ContainerType_Vector_USINT) *)
		nMaxIterations	:	UDINT;	(* Maximum number of iterations *)
		fConfidence	:	LREAL;	(* Confidence (0..1) *)
		nRefineIters	:	UDINT;	(* Maximum number of iterations of Levenberg-Marquardt algorithm to refine further the affine transform (using only inliers). Set to 0 to disable refining. *)
		hrPrev	:	HRESULT;	(* HRESULT indicating the result of previous operations (If SUCCEEDED(hrPrev) equals false, no operation is executed.) *)
	END_VAR

END_FUNCTION

// Functions/Geometric and Coordinate Transformations/F_VN_GetPerspectiveTransformation

